C07259=1059.763,-17.708,-67.702,171.487,27.976,155.219
C07260=1059.770,-17.459,-67.715,171.489,27.977,155.219
C07261=1059.775,-17.210,-67.729,171.490,27.980,155.219
C07262=1059.782,-16.960,-67.743,171.492,27.982,155.219
C07263=1059.788,-16.710,-67.756,171.493,27.984,155.220
C07264=1059.794,-16.461,-67.771,171.495,27.986,155.220
C07265=1059.801,-16.211,-67.784,171.497,27.989,155.220
C07266=1059.806,-15.962,-67.798,171.498,27.991,155.220
C07267=1059.813,-15.712,-67.812,171.500,27.993,155.221
C07268=1059.818,-15.462,-67.825,171.502,27.995,155.221
C07269=1059.825,-15.214,-67.839,171.502,27.997,155.221
C07270=1059.831,-14.963,-67.854,171.504,27.999,155.221
C07271=1059.837,-14.714,-67.867,171.506,28.002,155.222
C07272=1059.843,-14.464,-67.881,171.507,28.004,155.222
C07273=1059.850,-14.215,-67.895,171.509,28.006,155.222
C07274=1059.855,-13.966,-67.909,171.510,28.009,155.223
C07275=1059.861,-13.715,-67.923,171.512,28.011,155.223
C07276=1059.868,-13.467,-67.937,171.514,28.013,155.223
C07277=1059.873,-13.217,-67.951,171.515,28.015,155.223
C07278=1059.880,-12.967,-67.965,171.517,28.018,155.224
C07279=1059.886,-12.718,-67.979,171.519,28.020,155.224
C07280=1059.892,-12.468,-67.994,171.520,28.022,155.224
C07281=1059.898,-12.219,-68.007,171.522,28.024,155.225
C07282=1059.904,-11.969,-68.021,171.523,28.026,155.225
C07283=1059.910,-11.719,-68.036,171.524,28.029,155.225
C07284=1059.916,-11.470,-68.049,171.526,28.031,155.225
C07285=1059.922,-11.220,-68.063,171.528,28.033,155.226
C07286=1059.928,-10.971,-68.078,171.529,28.035,155.226
C07287=1059.934,-10.722,-68.091,171.531,28.038,155.226
C07288=1059.941,-10.472,-68.106,171.532,28.040,155.226
C07289=1059.946,-10.222,-68.120,171.534,28.042,155.227
C07290=1059.953,-9.972,-68.133,171.536,28.045,155.227
C07291=1059.959,-9.723,-68.148,171.537,28.047,155.227
C07292=1059.965,-9.473,-68.162,171.539,28.049,155.228
C07293=1059.972,-9.225,-68.176,171.540,28.051,155.228
C07294=1059.977,-8.975,-68.190,171.541,28.054,155.228
C07295=1059.983,-8.725,-68.204,171.543,28.056,155.228
C07296=1059.990,-8.476,-68.218,171.545,28.058,155.229
C07297=1059.996,-8.226,-68.233,171.546,28.060,155.229
C07298=1060.001,-7.977,-68.247,171.548,28.063,155.229
C07299=1060.008,-7.727,-68.261,171.549,28.065,155.230
C07300=1060.014,-7.478,-68.275,171.551,28.067,155.230
C07301=1060.020,-7.228,-68.290,171.553,28.069,155.230
C07302=1060.027,-6.979,-68.304,171.554,28.072,155.230
C07303=1060.033,-6.729,-68.318,171.556,28.074,155.231
C07304=1060.039,-6.480,-68.332,171.557,28.076,155.231
C07305=1060.045,-6.229,-68.347,171.558,28.079,155.231
C07306=1060.051,-5.981,-68.361,171.560,28.081,155.232
C07307=1060.057,-5.731,-68.375,171.562,28.083,155.232
C07308=1060.063,-5.482,-68.389,171.563,28.085,155.232
C07309=1060.070,-5.232,-68.403,171.565,28.088,155.232
C07310=1060.076,-4.983,-68.418,171.566,28.090,155.233
C07311=1060.082,-4.732,-68.432,171.568,28.092,155.233
C07312=1060.088,-4.484,-68.446,171.570,28.094,155.233
C07313=1060.095,-4.234,-68.461,171.571,28.097,155.233
C07314=1060.101,-3.984,-68.475,171.573,28.099,155.234
C07315=1060.106,-3.735,-68.490,171.574,28.101,155.234
C07316=1060.113,-3.485,-68.503,171.575,28.104,155.234
C07317=1060.119,-3.236,-68.518,171.577,28.106,155.235
C07318=1060.125,-2.986,-68.533,171.579,28.108,155.235
C07319=1060.131,-2.737,-68.547,171.580,28.110,155.235
C07320=1060.137,-2.455,-68.563,171.582,28.113,155.236
C07321=1060.145,-2.174,-68.580,171.583,28.116,155.236
C07322=1060.151,-1.893,-68.596,171.585,28.118,155.236
C07323=1060.158,-1.612,-68.612,171.587,28.121,155.237
C07324=1060.164,-1.362,-68.627,171.588,28.123,155.237
C07325=1060.170,-1.113,-68.641,171.590,28.126,155.237
C07326=1060.176,-0.863,-68.656,171.591,28.128,155.238
C07327=1060.182,-0.614,-68.670,171.593,28.131,155.238
C07328=1060.188,-0.364,-68.685,171.595,28.134,155.238
C07329=1060.194,-0.114,-68.699,171.596,28.136,155.239
C07330=1060.200,0.135,-68.714,171.598,28.138,155.239
C07331=1060.207,0.385,-68.729,171.600,28.140,155.239
C07332=1060.212,0.634,-68.743,171.600,28.143,155.239
C07333=1060.218,0.884,-68.758,171.602,28.145,155.240
C07334=1060.224,1.133,-68.772,171.603,28.147,155.240
C07335=1060.231,1.383,-68.787,171.605,28.150,155.240
C07336=1060.236,1.632,-68.802,171.607,28.152,155.241
C07337=1060.243,1.882,-68.816,171.608,28.155,155.241
C07338=1060.248,2.131,-68.831,171.610,28.157,155.241
C07339=1060.254,2.381,-68.846,171.612,28.160,155.242
C07340=1060.260,2.630,-68.861,171.612,28.162,155.242
C07341=1060.266,2.879,-68.876,171.614,28.164,155.242
C07342=1060.272,3.130,-68.890,171.615,28.166,155.242
C07343=1060.278,3.379,-68.904,171.617,28.169,155.243
C07344=1060.284,3.628,-68.919,171.619,28.171,155.243
C07345=1060.291,3.878,-68.934,171.620,28.173,155.243
C07346=1060.297,4.127,-68.949,171.622,28.176,155.244
C07347=1060.303,4.377,-68.964,171.624,28.179,155.244
C07348=1060.309,4.626,-68.979,171.625,28.181,155.244
C07349=1060.315,4.876,-68.993,171.626,28.183,155.245
C07350=1060.321,5.125,-69.008,171.627,28.186,155.245
C07351=1060.327,5.374,-69.022,171.629,28.188,155.245
C07352=1060.333,5.624,-69.037,171.631,28.190,155.246
C07353=1060.340,5.874,-69.052,171.632,28.193,155.246
C07354=1060.345,6.123,-69.067,171.634,28.195,155.246
C07355=1060.352,6.372,-69.082,171.636,28.197,155.246
C07356=1060.358,6.622,-69.097,171.637,28.200,155.247
C07357=1060.364,6.871,-69.111,171.638,28.202,155.247
C07358=1060.370,7.121,-69.127,171.640,28.204,155.247
C07359=1060.376,7.371,-69.142,171.641,28.207,155.248
C07360=1060.382,7.620,-69.156,171.643,28.209,155.248
C07361=1060.388,7.870,-69.170,171.644,28.212,155.248
C07362=1060.394,8.119,-69.185,171.646,28.214,155.249
C07363=1060.400,8.368,-69.200,171.648,28.217,155.249
C07364=1060.406,8.618,-69.215,171.648,28.219,155.249
C07365=1060.413,8.868,-69.230,171.650,28.221,155.250
C07366=1060.419,9.117,-69.245,171.652,28.224,155.250
C07367=1060.425,9.366,-69.259,171.653,28.226,155.250
C07368=1060.431,9.616,-69.274,171.655,28.228,155.251
C07369=1060.438,9.866,-69.289,171.656,28.231,155.251
C07370=1060.444,10.115,-69.306,171.658,28.233,155.251
C07371=1060.450,10.364,-69.320,171.660,28.236,155.251
C07372=1060.456,10.614,-69.335,171.660,28.238,155.252
C07373=1060.462,10.863,-69.350,171.662,28.240,155.252
C07374=1060.468,11.112,-69.365,171.664,28.243,155.252
C07375=1060.474,11.362,-69.380,171.665,28.245,155.253
C07376=1060.481,11.612,-69.395,171.667,28.248,155.253
C07377=1060.487,11.861,-69.409,171.669,28.250,155.253
C07378=1060.493,12.111,-69.425,171.670,28.252,155.254
C07379=1060.499,12.360,-69.440,171.671,28.255,155.254
C07380=1060.505,12.610,-69.455,171.672,28.257,155.254
C07381=1060.511,12.859,-69.469,171.674,28.259,155.255
C07382=1060.518,13.109,-69.485,171.676,28.262,155.255
C07383=1060.524,13.357,-69.500,171.677,28.264,155.255
C07384=1060.531,13.642,-69.517,171.679,28.267,155.256
C07385=1060.538,13.925,-69.534,171.681,28.269,155.256
C07386=1060.546,14.208,-69.551,171.682,28.272,155.256
C07387=1060.552,14.491,-69.568,171.684,28.275,155.257
C07388=1060.559,14.740,-69.584,171.685,28.277,155.257
C07389=1060.564,14.990,-69.599,171.687,28.280,155.257
C07390=1060.570,15.239,-69.614,171.689,28.282,155.258
C07391=1060.576,15.489,-69.629,171.690,28.285,155.258
C07392=1060.582,15.739,-69.644,171.692,28.287,155.258
C07393=1060.588,15.987,-69.660,171.693,28.290,155.259
C07394=1060.595,16.237,-69.675,171.694,28.292,155.259
C07395=1060.600,16.487,-69.690,171.696,28.295,155.259
C07396=1060.607,16.737,-69.705,171.697,28.297,155.260
C07397=1060.613,16.986,-69.721,171.699,28.299,155.260
C07398=1060.618,17.235,-69.736,171.701,28.302,155.260
C07399=1060.625,17.485,-69.751,171.702,28.304,155.261
C07400=1060.631,17.734,-69.766,171.703,28.307,155.261
C07401=1060.637,17.984,-69.782,171.705,28.309,155.261
C07402=1060.643,18.233,-69.797,171.706,28.312,155.262
C07403=1060.648,18.483,-69.812,171.708,28.314,155.262
C07404=1060.655,18.732,-69.828,171.709,28.317,155.262
C07405=1060.662,18.981,-69.843,171.711,28.319,155.263
C07406=1060.667,19.231,-69.858,171.713,28.321,155.263
C07407=1060.674,19.480,-69.874,171.713,28.324,155.263
C07408=1060.680,19.730,-69.889,171.715,28.326,155.264
C07409=1060.685,19.979,-69.904,171.716,28.329,155.264
C07410=1060.692,20.228,-69.920,171.718,28.331,155.264
C07411=1060.698,20.478,-69.935,171.720,28.334,155.265
C07412=1060.704,20.728,-69.950,171.721,28.336,155.265
C07413=1060.710,20.977,-69.967,171.722,28.339,155.265
C07414=1060.716,21.227,-69.981,171.724,28.341,155.266
C07415=1060.722,21.476,-69.998,171.725,28.344,155.266
C07416=1060.728,21.725,-70.012,171.727,28.346,155.266
C07417=1060.734,21.974,-70.029,171.728,28.349,155.267
C07418=1060.740,22.224,-70.044,171.730,28.351,155.267
C07419=1060.746,22.474,-70.059,171.732,28.354,155.267
C07420=1060.753,22.723,-70.075,171.732,28.356,155.268
C07421=1060.758,22.973,-70.090,171.734,28.359,155.268
C07422=1060.765,23.222,-70.106,171.736,28.361,155.268
C07423=1060.770,23.471,-70.121,171.737,28.364,155.269
C07424=1060.777,23.720,-70.137,171.739,28.366,155.269
C07425=1060.782,23.970,-70.152,171.741,28.369,155.269
C07426=1060.789,24.219,-70.168,171.741,28.371,155.270
C07427=1060.795,24.469,-70.184,171.743,28.374,155.270
C07428=1060.801,24.718,-70.199,171.744,28.376,155.270
C07429=1060.807,24.968,-70.215,171.746,28.379,155.271
C07430=1060.814,25.217,-70.230,171.748,28.381,155.271
C07431=1060.819,25.467,-70.246,171.749,28.384,155.271
C07432=1060.825,25.717,-70.262,171.750,28.386,155.272
C07433=1060.831,25.966,-70.277,171.752,28.388,155.272
C07434=1060.837,26.215,-70.293,171.753,28.391,155.272
C07435=1060.844,26.465,-70.308,171.755,28.393,155.273
C07436=1060.849,26.714,-70.324,171.756,28.396,155.273
C07437=1060.856,26.963,-70.340,171.758,28.398,155.273
C07438=1060.862,27.213,-70.355,171.759,28.400,155.274
C07439=1060.868,27.462,-70.372,171.760,28.403,155.274
C07440=1060.874,27.712,-70.387,171.762,28.406,155.275
C07441=1060.880,27.961,-70.403,171.764,28.408,155.275
C07442=1060.887,28.210,-70.419,171.765,28.411,155.275
C07443=1060.892,28.460,-70.434,171.767,28.413,155.275
C07444=1060.898,28.710,-70.450,171.768,28.416,155.276
C07445=1060.905,28.959,-70.466,171.769,28.418,155.276
C07446=1060.911,29.209,-70.482,171.771,28.421,155.277
C07447=1060.917,29.458,-70.498,171.772,28.423,155.277
C07448=1060.924,29.743,-70.515,171.774,28.426,155.277
C07449=1060.930,30.027,-70.534,171.776,28.429,155.278
C07450=1060.938,30.312,-70.551,171.777,28.432,155.278
C07451=1060.944,30.596,-70.570,171.779,28.435,155.279
C07452=1060.950,30.846,-70.586,171.780,28.438,155.279
C07453=1060.956,31.096,-70.602,171.782,28.440,155.279
C07454=1060.962,31.345,-70.617,171.784,28.443,155.280
C07455=1060.968,31.594,-70.634,171.785,28.445,155.280
C07456=1060.974,31.844,-70.649,171.786,28.447,155.280
C07457=1060.980,32.093,-70.666,171.787,28.450,155.281
C07458=1060.987,32.342,-70.681,171.789,28.452,155.281
C07459=1060.993,32.592,-70.697,171.791,28.455,155.281
C07460=1060.998,32.842,-70.713,171.792,28.458,155.282
C07461=1061.004,33.091,-70.729,171.794,28.460,155.282
C07462=1061.011,33.340,-70.745,171.795,28.463,155.282
C07463=1061.017,33.589,-70.761,171.796,28.465,155.283
C07464=1061.023,33.839,-70.777,171.798,28.468,155.283
C07465=1061.028,34.089,-70.793,171.799,28.470,155.283
C07466=1061.035,34.338,-70.809,171.801,28.473,155.284
C07467=1061.041,34.587,-70.825,171.803,28.476,155.284
C07468=1061.047,34.836,-70.841,171.803,28.478,155.284
C07469=1061.053,35.086,-70.857,171.805,28.480,155.285
C07470=1061.059,35.335,-70.874,171.807,28.483,155.285
C07471=1061.065,35.585,-70.889,171.808,28.485,155.286
C07472=1061.071,35.834,-70.905,171.810,28.488,155.286
C07473=1061.077,36.083,-70.921,171.812,28.490,155.286
C07474=1061.083,36.333,-70.937,171.812,28.493,155.287
C07475=1061.089,36.582,-70.954,171.814,28.495,155.287
C07476=1061.096,36.831,-70.969,171.815,28.498,155.287
C07477=1061.102,37.081,-70.986,171.817,28.501,155.288
C07478=1061.108,37.331,-71.002,171.819,28.503,155.288
C07479=1061.114,37.580,-71.018,171.820,28.506,155.288
C07480=1061.120,37.829,-71.035,171.821,28.508,155.289
C07481=1061.126,38.079,-71.050,171.823,28.511,155.289
C07482=1061.132,38.329,-71.066,171.824,28.513,155.289
C07483=1061.138,38.578,-71.083,171.826,28.516,155.290
C07484=1061.144,38.827,-71.099,171.827,28.518,155.290
C07485=1061.150,39.077,-71.115,171.828,28.521,155.291
C07486=1061.156,39.326,-71.132,171.830,28.523,155.291
C07487=1061.162,39.575,-71.148,171.831,28.526,155.291
C07488=1061.168,39.825,-71.164,171.833,28.529,155.292
C07489=1061.173,40.074,-71.180,171.835,28.532,155.292
C07490=1061.179,40.323,-71.197,171.836,28.534,155.292
C07491=1061.185,40.573,-71.213,171.837,28.536,155.293
C07492=1061.192,40.823,-71.229,171.838,28.539,155.293
C07493=1061.198,41.072,-71.246,171.840,28.541,155.293
C07494=1061.204,41.321,-71.263,171.842,28.544,155.294
C07495=1061.210,41.570,-71.279,171.843,28.547,155.294
C07496=1061.216,41.820,-71.295,171.844,28.549,155.294
C07497=1061.222,42.069,-71.311,171.846,28.552,155.295
C07498=1061.228,42.318,-71.328,171.847,28.555,155.295
C07499=1061.234,42.568,-71.344,171.849,28.557,155.296
C07500=1061.240,42.817,-71.360,171.851,28.560,155.296
C07501=1061.246,43.067,-71.377,171.852,28.562,155.296
C07502=1061.252,43.316,-71.393,171.853,28.564,155.297
C07503=1061.258,43.566,-71.409,171.854,28.567,155.297
C07504=1061.264,43.815,-71.426,171.856,28.570,155.297
C07505=1061.270,44.064,-71.443,171.858,28.573,155.298
C07506=1061.276,44.313,-71.459,171.859,28.575,155.298
C07507=1061.282,44.563,-71.476,171.860,28.577,155.299
C07508=1061.288,44.812,-71.492,171.862,28.580,155.299
C07509=1061.294,45.062,-71.509,171.863,28.583,155.299
C07510=1061.300,45.312,-71.525,171.865,28.586,155.300
C07511=1061.306,45.561,-71.542,171.866,28.588,155.300
C07512=1061.312,45.845,-71.561,171.868,28.591,155.300
C07513=1061.319,46.130,-71.580,171.870,28.594,155.301
C07514=1061.326,46.414,-71.599,171.871,28.597,155.301
C07515=1061.333,46.699,-71.618,171.873,28.600,155.302
C07516=1061.339,46.948,-71.634,171.874,28.603,155.302
C07517=1061.344,47.198,-71.651,171.876,28.605,155.302
C07518=1061.350,47.447,-71.668,171.877,28.608,155.303
C07519=1061.356,47.696,-71.684,171.878,28.611,155.303
C07520=1061.362,47.946,-71.701,171.880,28.613,155.304
C07521=1061.368,48.196,-71.717,171.881,28.616,155.304
C07522=1061.374,48.444,-71.734,171.883,28.618,155.304
C07523=1061.380,48.694,-71.751,171.885,28.621,155.305
C07524=1061.385,48.943,-71.767,171.885,28.624,155.305
C07525=1061.392,49.192,-71.784,171.887,28.627,155.306
C07526=1061.398,49.442,-71.801,171.889,28.629,155.306
C07527=1061.404,49.691,-71.817,171.890,28.632,155.306
C07528=1061.410,49.940,-71.835,171.892,28.634,155.307
C07529=1061.416,50.190,-71.851,171.892,28.637,155.307
C07530=1061.422,50.439,-71.867,171.894,28.639,155.307
C07531=1061.428,50.689,-71.885,171.896,28.642,155.308
C07532=1061.434,50.938,-71.902,171.897,28.645,155.308
C07533=1061.440,51.188,-71.918,171.899,28.647,155.309
C07534=1061.445,51.437,-71.935,171.900,28.650,155.309
C07535=1061.452,51.687,-71.952,171.901,28.652,155.309
C07536=1061.458,51.935,-71.969,171.903,28.655,155.310
C07537=1061.464,52.185,-71.985,171.905,28.658,155.310
C07538=1061.469,52.434,-72.002,171.906,28.661,155.310
C07539=1061.475,52.683,-72.019,171.908,28.663,155.311
C07540=1061.482,52.933,-72.036,171.908,28.665,155.311
C07541=1061.487,53.182,-72.053,171.910,28.668,155.311
C07542=1061.493,53.432,-72.070,171.912,28.671,155.312
C07543=1061.500,53.681,-72.087,171.913,28.673,155.312
C07544=1061.505,53.931,-72.104,171.915,28.676,155.313
C07545=1061.512,54.179,-72.121,171.916,28.678,155.313
C07546=1061.518,54.429,-72.137,171.917,28.681,155.313
C07547=1061.523,54.679,-72.154,171.919,28.683,155.314
C07548=1061.530,54.928,-72.171,171.921,28.686,155.314
C07549=1061.536,55.177,-72.187,171.922,28.689,155.314
C07550=1061.542,55.427,-72.205,171.924,28.692,155.315
C07551=1061.548,55.676,-72.222,171.924,28.694,155.315
C07552=1061.554,55.925,-72.239,171.926,28.697,155.316
C07553=1061.560,56.174,-72.256,171.928,28.699,155.316
C07554=1061.566,56.424,-72.273,171.929,28.702,155.316
C07555=1061.572,56.673,-72.290,171.931,28.704,155.317
C07556=1061.578,56.923,-72.307,171.932,28.707,155.317
C07557=1061.584,57.172,-72.324,171.933,28.710,155.317
C07558=1061.590,57.421,-72.340,171.935,28.712,155.318
C07559=1061.596,57.670,-72.358,171.937,28.715,155.318
C07560=1061.602,57.920,-72.374,171.938,28.717,155.319
C07561=1061.608,58.169,-72.392,171.940,28.720,155.319
C07562=1061.614,58.418,-72.409,171.940,28.723,155.319
C07563=1061.621,58.668,-72.426,171.942,28.725,155.320
C07564=1061.626,58.917,-72.443,171.944,28.728,155.320
C07565=1061.633,59.167,-72.460,171.945,28.730,155.320
C07566=1061.639,59.416,-72.477,171.947,28.733,155.321
C07567=1061.645,59.665,-72.494,171.948,28.735,155.321
C07568=1061.651,59.915,-72.511,171.949,28.738,155.322
C07569=1061.657,60.164,-72.528,171.951,28.741,155.322
C07570=1061.664,60.414,-72.546,171.953,28.743,155.322
C07571=1061.669,60.663,-72.562,171.954,28.746,155.323
C07572=1061.675,60.912,-72.580,171.956,28.748,155.323
C07573=1061.682,61.161,-72.597,171.957,28.750,155.323
C07574=1061.688,61.411,-72.613,171.958,28.753,155.324
C07575=1061.694,61.660,-72.631,171.960,28.756,155.324
C07576=1061.701,61.944,-72.650,171.961,28.759,155.324
C07577=1061.708,62.228,-72.670,171.963,28.762,155.325
C07578=1061.715,62.514,-72.690,171.965,28.765,155.325
C07579=1061.721,62.797,-72.709,171.966,28.768,155.326
C07580=1061.728,63.047,-72.726,171.968,28.770,155.326
C07581=1061.734,63.296,-72.744,171.970,28.773,155.326
C07582=1061.740,63.546,-72.761,171.971,28.775,155.327
C07583=1061.747,63.794,-72.778,171.973,28.778,155.327
C07584=1061.753,64.044,-72.796,171.974,28.780,155.328
C07585=1061.759,64.293,-72.812,171.975,28.783,155.328
C07586=1061.765,64.543,-72.830,171.977,28.786,155.328
C07587=1061.770,64.792,-72.847,171.978,28.788,155.329
C07588=1061.776,65.041,-72.864,171.980,28.791,155.329
C07589=1061.783,65.291,-72.882,171.982,28.793,155.329
C07590=1061.789,65.539,-72.899,171.982,28.796,155.330
C07591=1061.795,65.789,-72.917,171.984,28.799,155.330
C07592=1061.800,66.039,-72.934,171.986,28.802,155.331
C07593=1061.807,66.288,-72.951,171.987,28.804,155.331
C07594=1061.813,66.537,-72.969,171.989,28.806,155.331
C07595=1061.818,66.786,-72.986,171.991,28.809,155.332
C07596=1061.825,67.036,-73.004,171.991,28.812,155.332
C07597=1061.830,67.285,-73.021,171.993,28.815,155.333
C07598=1061.837,67.535,-73.039,171.994,28.817,155.333
C07599=1061.843,67.783,-73.056,171.996,28.820,155.333
C07600=1061.849,68.033,-73.074,171.998,28.822,155.334
C07601=1061.854,68.283,-73.091,171.999,28.825,155.334
C07602=1061.860,68.532,-73.109,172.000,28.828,155.334
C07603=1061.867,68.781,-73.126,172.002,28.830,155.335
C07604=1061.873,69.031,-73.144,172.003,28.833,155.335
C07605=1061.878,69.280,-73.161,172.005,28.835,155.336
C07606=1061.885,69.529,-73.179,172.007,28.838,155.336
C07607=1061.891,69.778,-73.196,172.007,28.841,155.336
C07608=1061.897,70.028,-73.214,172.009,28.843,155.337
C07609=1061.902,70.277,-73.232,172.010,28.846,155.337
C07610=1061.908,70.526,-73.249,172.012,28.848,155.337
C07611=1061.915,70.776,-73.267,172.014,28.851,155.338
C07612=1061.920,71.025,-73.284,172.015,28.854,155.338
C07613=1061.926,71.274,-73.302,172.016,28.856,155.339
C07614=1061.932,71.523,-73.320,172.018,28.859,155.339
C07615=1061.938,71.773,-73.338,172.019,28.862,155.339
C07616=1061.944,72.022,-73.355,172.021,28.865,155.340
C07617=1061.950,72.272,-73.373,172.023,28.867,155.340
C07618=1061.956,72.520,-73.391,172.024,28.870,155.341
C07619=1061.962,72.770,-73.409,172.025,28.872,155.341
C07620=1061.968,73.019,-73.426,172.027,28.875,155.341
C07621=1061.974,73.269,-73.444,172.028,28.878,155.342
C07622=1061.979,73.518,-73.462,172.030,28.881,155.342
C07623=1061.986,73.767,-73.479,172.031,28.883,155.343
C07624=1061.992,74.016,-73.497,172.032,28.886,155.343
C07625=1061.998,74.266,-73.515,172.034,28.888,155.343
C07626=1062.004,74.516,-73.533,172.035,28.891,155.344
C07627=1062.010,74.764,-73.551,172.037,28.894,155.344
C07628=1062.016,75.014,-73.569,172.039,28.896,155.344
C07629=1062.021,75.263,-73.586,172.040,28.899,155.345
C07630=1062.028,75.513,-73.604,172.041,28.902,155.345
C07631=1062.034,75.761,-73.621,172.043,28.904,155.346
C07632=1062.040,76.011,-73.639,172.044,28.907,155.346
C07633=1062.046,76.259,-73.658,172.046,28.909,155.346
C07634=1062.052,76.509,-73.676,172.048,28.912,155.347
C07635=1062.058,76.759,-73.693,172.049,28.915,155.347
C07636=1062.064,77.008,-73.711,172.050,28.917,155.348
C07637=1062.070,77.258,-73.729,172.052,28.920,155.348
C07638=1062.075,77.506,-73.747,172.053,28.922,155.348
C07639=1062.082,77.756,-73.765,172.055,28.925,155.349
C07640=1062.088,78.040,-73.785,172.056,28.928,155.349
C07641=1062.096,78.324,-73.806,172.058,28.931,155.350
C07642=1062.102,78.608,-73.826,172.060,28.934,155.350
C07643=1062.109,78.892,-73.847,172.061,28.937,155.351
C07644=1062.115,79.142,-73.865,172.063,28.940,155.351
C07645=1062.121,79.391,-73.882,172.065,28.943,155.351
C07646=1062.126,79.641,-73.901,172.066,28.946,155.352
C07647=1062.132,79.890,-73.920,172.068,28.948,155.352
C07648=1062.138,80.139,-73.937,172.068,28.951,155.353
C07649=1062.144,80.389,-73.955,172.070,28.953,155.353
C07650=1062.150,80.637,-73.973,172.072,28.956,155.353
C07651=1062.156,80.887,-73.991,172.073,28.959,155.354
C07652=1062.162,81.135,-74.010,172.075,28.961,155.354
C07653=1062.168,81.385,-74.027,172.077,28.964,155.354
C07654=1062.173,81.635,-74.046,172.077,28.967,155.355
C07655=1062.179,81.884,-74.064,172.079,28.969,155.355
C07656=1062.185,82.133,-74.082,172.081,28.972,155.356
C07657=1062.191,82.383,-74.100,172.082,28.975,155.356
C07658=1062.197,82.631,-74.118,172.084,28.978,155.356
C07659=1062.203,82.881,-74.136,172.086,28.980,155.357
C07660=1062.209,83.130,-74.155,172.086,28.983,155.357
C07661=1062.215,83.380,-74.173,172.088,28.985,155.358
C07662=1062.221,83.629,-74.192,172.090,28.988,155.358
C07663=1062.227,83.878,-74.209,172.091,28.991,155.358
C07664=1062.233,84.128,-74.227,172.093,28.993,155.359
C07665=1062.239,84.377,-74.246,172.095,28.996,155.359
C07666=1062.245,84.626,-74.264,172.095,28.999,155.360
C07667=1062.250,84.875,-74.283,172.097,29.001,155.360
C07668=1062.256,85.125,-74.301,172.098,29.004,155.360
C07669=1062.262,85.373,-74.319,172.100,29.007,155.361
C07670=1062.268,85.623,-74.337,172.102,29.009,155.361
C07671=1062.275,85.872,-74.356,172.103,29.012,155.361
C07672=1062.280,86.121,-74.373,172.105,29.015,155.362
C07673=1062.286,86.371,-74.392,172.106,29.017,155.362
C07674=1062.292,86.620,-74.410,172.107,29.020,155.363
C07675=1062.299,86.870,-74.429,172.109,29.023,155.363
C07676=1062.304,87.118,-74.447,172.111,29.025,155.364
C07677=1062.310,87.368,-74.465,172.112,29.028,155.364
C07678=1062.317,87.617,-74.484,172.114,29.030,155.364
C07679=1062.322,87.866,-74.502,172.116,29.033,155.365
C07680=1062.328,88.115,-74.521,172.116,29.036,155.365
C07681=1062.334,88.365,-74.539,172.118,29.038,155.365
C07682=1062.341,88.614,-74.557,172.120,29.041,155.366
C07683=1062.346,88.863,-74.575,172.121,29.044,155.366
C07684=1062.352,89.113,-74.594,172.123,29.047,155.367
C07685=1062.358,89.362,-74.613,172.125,29.049,155.367
C07686=1062.365,89.611,-74.631,172.125,29.051,155.367
C07687=1062.370,89.860,-74.649,172.127,29.054,155.368
C07688=1062.376,90.109,-74.668,172.129,29.057,155.368
C07689=1062.382,90.358,-74.687,172.130,29.060,155.369
C07690=1062.388,90.608,-74.705,172.132,29.062,155.369
C07691=1062.394,90.857,-74.723,172.134,29.065,155.369
C07692=1062.400,91.106,-74.742,172.135,29.068,155.370
C07693=1062.406,91.356,-74.760,172.136,29.070,155.370
C07694=1062.412,91.605,-74.779,172.138,29.073,155.371
C07695=1062.418,91.854,-74.798,172.139,29.076,155.371
C07696=1062.424,92.103,-74.816,172.141,29.078,155.371
C07697=1062.429,92.353,-74.835,172.143,29.081,155.372
C07698=1062.436,92.602,-74.854,172.144,29.084,155.372
C07699=1062.441,92.851,-74.872,172.146,29.086,155.372
C07700=1062.447,93.100,-74.890,172.147,29.089,155.373
C07701=1062.453,93.350,-74.910,172.148,29.092,155.373
C07702=1062.459,93.599,-74.928,172.150,29.094,155.374
C07703=1062.464,93.848,-74.947,172.151,29.097,155.374
C07704=1062.471,94.132,-74.968,172.153,29.100,155.375
C07705=1062.479,94.416,-74.989,172.155,29.103,155.375
C07706=1062.485,94.701,-75.011,172.156,29.107,155.376
C07707=1062.492,94.985,-75.032,172.158,29.109,155.376
C07708=1062.498,95.234,-75.051,172.160,29.112,155.376
C07709=1062.504,95.482,-75.070,172.161,29.115,155.377
C07710=1062.509,95.732,-75.088,172.163,29.117,155.377
C07711=1062.515,95.982,-75.107,172.164,29.120,155.378
C07712=1062.521,96.231,-75.126,172.166,29.123,155.378
C07713=1062.527,96.480,-75.145,172.168,29.126,155.378
C07714=1062.533,96.729,-75.164,172.169,29.128,155.379
C07715=1062.539,96.978,-75.182,172.170,29.131,155.379
C07716=1062.545,97.227,-75.201,172.172,29.133,155.379
C07717=1062.551,97.477,-75.220,172.174,29.136,155.380
C07718=1062.557,97.726,-75.239,172.175,29.139,155.380
C07719=1062.563,97.976,-75.257,172.177,29.141,155.381
C07720=1062.569,98.225,-75.277,172.178,29.144,155.381
C07721=1062.574,98.474,-75.295,172.180,29.147,155.381
C07722=1062.580,98.723,-75.314,172.182,29.150,155.382
C07723=1062.587,98.972,-75.333,172.182,29.152,155.382
C07724=1062.592,99.222,-75.352,172.184,29.155,155.383
C07725=1062.599,99.471,-75.371,172.186,29.158,155.383
C07726=1062.604,99.720,-75.390,172.187,29.160,155.384
C07727=1062.611,99.969,-75.408,172.189,29.163,155.384
C07728=1062.616,100.219,-75.428,172.191,29.165,155.384
C07729=1062.622,100.467,-75.446,172.192,29.168,155.385
C07730=1062.628,100.717,-75.465,172.194,29.171,155.385
C07731=1062.634,100.966,-75.484,172.195,29.173,155.385
C07732=1062.640,101.215,-75.503,172.196,29.176,155.386
C07733=1062.646,101.465,-75.522,172.198,29.179,155.386
C07734=1062.652,101.714,-75.541,172.200,29.182,155.387
C07735=1062.658,101.963,-75.560,172.201,29.184,155.387
C07736=1062.664,102.213,-75.580,172.203,29.187,155.387
C07737=1062.669,102.461,-75.599,172.205,29.190,155.388
C07738=1062.675,102.710,-75.618,172.206,29.192,155.388
C07739=1062.681,102.959,-75.637,172.207,29.195,155.389
C07740=1062.687,103.209,-75.656,172.209,29.198,155.389
C07741=1062.692,103.458,-75.676,172.210,29.200,155.390
C07742=1062.699,103.707,-75.694,172.212,29.203,155.390
C07743=1062.705,103.957,-75.713,172.214,29.206,155.390
C07744=1062.710,104.206,-75.733,172.215,29.209,155.391
C07745=1062.716,104.455,-75.753,172.217,29.211,155.391
C07746=1062.723,104.704,-75.771,172.219,29.214,155.392
C07747=1062.728,104.953,-75.790,172.220,29.217,155.392
C07748=1062.733,105.202,-75.809,172.221,29.219,155.392
C07749=1062.739,105.452,-75.829,172.223,29.222,155.393
C07750=1062.746,105.701,-75.847,172.224,29.225,155.393
C07751=1062.752,105.949,-75.867,172.226,29.228,155.394
C07752=1062.757,106.199,-75.886,172.228,29.230,155.394
C07753=1062.763,106.448,-75.906,172.229,29.233,155.394
C07754=1062.769,106.697,-75.924,172.231,29.235,155.395
C07755=1062.775,106.946,-75.944,172.233,29.238,155.395
C07756=1062.781,107.196,-75.964,172.234,29.241,155.395
C07757=1062.787,107.445,-75.983,172.235,29.243,155.396
C07758=1062.792,107.695,-76.002,172.237,29.246,155.396
C07759=1062.799,107.943,-76.021,172.238,29.249,155.397
C07760=1062.805,108.193,-76.041,172.240,29.251,155.397
C07761=1062.811,108.442,-76.060,172.242,29.254,155.398
C07762=1062.816,108.691,-76.079,172.243,29.257,155.398
C07763=1062.823,108.940,-76.099,172.245,29.260,155.398
C07764=1062.829,109.189,-76.118,172.247,29.262,155.399
C07765=1062.834,109.439,-76.137,172.248,29.265,155.399
C07766=1062.840,109.688,-76.157,172.250,29.268,155.400
C07767=1062.846,109.937,-76.176,172.251,29.270,155.400
C07768=1062.853,110.221,-76.199,172.253,29.273,155.400
C07769=1062.860,110.505,-76.220,172.255,29.277,155.401
C07770=1062.867,110.789,-76.242,172.257,29.279,155.401
C07771=1062.874,111.074,-76.264,172.258,29.283,155.402
C07772=1062.879,111.323,-76.284,172.260,29.285,155.402
C07773=1062.885,111.572,-76.303,172.262,29.288,155.402
C07774=1062.891,111.821,-76.323,172.263,29.290,155.403
C07775=1062.897,112.070,-76.343,172.265,29.293,155.403
C07776=1062.903,112.319,-76.363,172.267,29.296,155.404
C07777=1062.909,112.569,-76.382,172.268,29.298,155.404
C07778=1062.914,112.818,-76.401,172.270,29.301,155.405
C07779=1062.920,113.067,-76.421,172.272,29.304,155.405
C07780=1062.926,113.316,-76.440,172.272,29.306,155.405
C07781=1062.932,113.565,-76.460,172.274,29.309,155.406
C07782=1062.938,113.814,-76.479,172.276,29.312,155.406
C07783=1062.944,114.063,-76.499,172.277,29.315,155.407
C07784=1062.949,114.313,-76.519,172.279,29.317,155.407
C07785=1062.955,114.562,-76.539,172.281,29.320,155.407
C07786=1062.961,114.811,-76.558,172.282,29.323,155.408
C07787=1062.967,115.060,-76.578,172.284,29.326,155.408
C07788=1062.973,115.309,-76.597,172.286,29.329,155.409
C07789=1062.979,115.558,-76.617,172.287,29.332,155.409
C07790=1062.984,115.808,-76.637,172.289,29.334,155.410
C07791=1062.990,116.057,-76.657,172.291,29.337,155.410
C07792=1062.996,116.306,-76.677,172.291,29.340,155.410
C07793=1063.001,116.555,-76.696,172.293,29.342,155.411
C07794=1063.007,116.804,-76.716,172.295,29.345,155.411
C07795=1063.013,117.053,-76.735,172.296,29.348,155.412
C07796=1063.018,117.302,-76.756,172.298,29.350,155.412
C07797=1063.024,117.551,-76.776,172.300,29.353,155.412
C07798=1063.030,117.801,-76.795,172.301,29.356,155.413
C07799=1063.036,118.050,-76.815,172.303,29.359,155.413
C07800=1063.042,118.299,-76.835,172.305,29.361,155.414
C07801=1063.047,118.549,-76.855,172.306,29.364,155.414
C07802=1063.053,118.797,-76.875,172.308,29.367,155.414
C07803=1063.059,119.046,-76.895,172.310,29.370,155.415
C07804=1063.065,119.296,-76.914,172.311,29.373,155.415
C07805=1063.071,119.545,-76.934,172.312,29.375,155.416
C07806=1063.076,119.794,-76.955,172.314,29.378,155.416
C07807=1063.082,120.043,-76.974,172.315,29.381,155.417
C07808=1063.088,120.292,-76.994,172.317,29.384,155.417
C07809=1063.095,120.541,-77.014,172.319,29.386,155.417
C07810=1063.100,120.791,-77.035,172.320,29.389,155.418
C07811=1063.106,121.040,-77.054,172.322,29.392,155.418
C07812=1063.112,121.289,-77.074,172.324,29.394,155.419
C07813=1063.118,121.538,-77.094,172.325,29.397,155.419
C07814=1063.123,121.787,-77.115,172.327,29.400,155.419
C07815=1063.128,122.036,-77.134,172.329,29.403,155.420
C07816=1063.135,122.286,-77.154,172.330,29.405,155.420
C07817=1063.141,122.534,-77.174,172.332,29.408,155.421
C07818=1063.147,122.783,-77.194,172.334,29.411,155.421
C07819=1063.152,123.032,-77.215,172.335,29.413,155.421
C07820=1063.158,123.282,-77.234,172.337,29.416,155.422
C07821=1063.164,123.531,-77.254,172.339,29.419,155.422
C07822=1063.171,123.780,-77.274,172.340,29.422,155.423
C07823=1063.176,124.029,-77.295,172.342,29.424,155.423
C07824=1063.182,124.278,-77.315,172.344,29.427,155.423
C07825=1063.188,124.527,-77.335,172.344,29.430,155.424
C07826=1063.193,124.777,-77.354,172.346,29.432,155.424
C07827=1063.199,125.026,-77.375,172.348,29.435,155.425
C07828=1063.205,125.275,-77.395,172.350,29.438,155.425
C07829=1063.211,125.524,-77.415,172.351,29.440,155.426
C07830=1063.217,125.773,-77.435,172.353,29.443,155.426
C07831=1063.223,126.022,-77.455,172.355,29.446,155.426
C07832=1063.230,126.306,-77.478,172.357,29.449,155.427
C07833=1063.237,126.590,-77.502,172.359,29.452,155.427
C07834=1063.244,126.875,-77.525,172.360,29.455,155.428
C07835=1063.249,127.158,-77.548,172.362,29.458,155.428
C07836=1063.255,127.407,-77.567,172.364,29.461,155.429
C07837=1063.262,127.657,-77.588,172.365,29.464,155.429
C07838=1063.268,127.906,-77.608,172.367,29.466,155.429
C07839=1063.273,128.155,-77.628,172.369,29.469,155.430
C07840=1063.280,128.404,-77.649,172.371,29.472,155.430
C07841=1063.286,128.653,-77.669,172.372,29.474,155.431
C07842=1063.291,128.902,-77.689,172.374,29.477,155.431
C07843=1063.297,129.151,-77.709,172.376,29.480,155.431
C07844=1063.304,129.401,-77.729,172.377,29.483,155.432
C07845=1063.309,129.650,-77.750,172.379,29.485,155.432
C07846=1063.315,129.898,-77.770,172.381,29.487,155.433
C07847=1063.322,130.148,-77.790,172.382,29.490,155.433
C07848=1063.327,130.397,-77.811,172.384,29.493,155.433
C07849=1063.333,130.646,-77.831,172.386,29.496,155.434
C07850=1063.339,130.895,-77.851,172.387,29.498,155.434
C07851=1063.345,131.144,-77.872,172.389,29.501,155.435
C07852=1063.351,131.393,-77.892,172.391,29.504,155.435
C07853=1063.358,131.642,-77.913,172.392,29.506,155.435
C07854=1063.363,131.891,-77.933,172.394,29.509,155.436
C07855=1063.369,132.140,-77.953,172.396,29.512,155.436
C07856=1063.375,132.390,-77.974,172.397,29.515,155.437
C07857=1063.381,132.639,-77.994,172.399,29.517,155.437
C07858=1063.386,132.888,-78.015,172.401,29.520,155.437
C07859=1063.392,133.136,-78.035,172.403,29.523,155.438
C07860=1063.398,133.386,-78.056,172.404,29.525,155.438
C07861=1063.403,133.635,-78.077,172.406,29.528,155.439
C07862=1063.409,133.884,-78.097,172.408,29.531,155.439
C07863=1063.415,134.134,-78.118,172.409,29.534,155.440
C07864=1063.421,134.382,-78.138,172.411,29.537,155.440
C07865=1063.427,134.631,-78.159,172.413,29.540,155.440
C07866=1063.433,134.881,-78.180,172.414,29.542,155.441
C07867=1063.439,135.130,-78.200,172.416,29.545,155.441
C07868=1063.444,135.378,-78.221,172.418,29.548,155.442
C07869=1063.451,135.628,-78.241,172.419,29.550,155.442
C07870=1063.456,135.877,-78.262,172.421,29.553,155.442
C07871=1063.462,136.125,-78.283,172.423,29.556,155.443
C07872=1063.468,136.375,-78.303,172.424,29.559,155.443
C07873=1063.473,136.624,-78.324,172.426,29.561,155.444
C07874=1063.480,136.874,-78.344,172.428,29.564,155.444
C07875=1063.486,137.122,-78.366,172.429,29.567,155.444
C07876=1063.491,137.371,-78.386,172.431,29.569,155.445
C07877=1063.498,137.620,-78.407,172.433,29.572,155.445
C07878=1063.503,137.869,-78.428,172.435,29.575,155.446
C07879=1063.508,138.118,-78.448,172.436,29.577,155.446
C07880=1063.515,138.367,-78.469,172.438,29.580,155.447
C07881=1063.520,138.616,-78.490,172.440,29.583,155.447
C07882=1063.526,138.866,-78.511,172.441,29.586,155.447
C07883=1063.532,139.115,-78.532,172.443,29.589,155.448
C07884=1063.538,139.363,-78.552,172.446,29.592,155.448
C07885=1063.544,139.613,-78.574,172.447,29.594,155.449
C07886=1063.549,139.862,-78.594,172.449,29.597,155.449
C07887=1063.556,140.111,-78.615,172.451,29.600,155.449
C07888=1063.561,140.360,-78.636,172.452,29.603,155.450
C07889=1063.567,140.610,-78.657,172.454,29.605,155.450
C07890=1063.573,140.858,-78.678,172.456,29.608,155.451
C07891=1063.578,141.107,-78.699,172.457,29.611,155.451
C07892=1063.585,141.356,-78.720,172.459,29.613,155.452
C07893=1063.590,141.605,-78.740,172.461,29.616,155.452
C07894=1063.596,141.854,-78.762,172.462,29.619,155.452
C07895=1063.602,142.104,-78.782,172.464,29.622,155.453
C07896=1063.608,142.388,-78.806,172.466,29.625,155.453
C07897=1063.615,142.672,-78.830,172.468,29.628,155.454
C07898=1063.622,142.956,-78.854,172.470,29.632,155.454
C07899=1063.628,143.239,-78.878,172.472,29.634,155.455
C07900=1063.634,143.488,-78.900,172.473,29.637,155.455
C07901=1063.640,143.737,-78.921,172.475,29.640,155.456
C07902=1063.645,143.987,-78.942,172.477,29.643,155.456
C07903=1063.651,144.235,-78.963,172.479,29.646,155.456
C07904=1063.658,144.485,-78.983,172.481,29.649,155.457
C07905=1063.663,144.733,-79.005,172.483,29.651,155.457
C07906=1063.669,144.982,-79.026,172.485,29.654,155.458
C07907=1063.675,145.231,-79.047,172.486,29.657,155.458
C07908=1063.681,145.481,-79.069,172.488,29.659,155.458
C07909=1063.686,145.730,-79.089,172.490,29.662,155.459
C07910=1063.692,145.979,-79.111,172.491,29.665,155.459
C07911=1063.698,146.228,-79.132,172.493,29.667,155.460
C07912=1063.705,146.476,-79.153,172.495,29.671,155.460
C07913=1063.710,146.726,-79.174,172.496,29.673,155.461
C07914=1063.716,146.975,-79.195,172.498,29.676,155.461
C07915=1063.722,147.223,-79.217,172.500,29.679,155.461
C07916=1063.728,147.473,-79.237,172.502,29.681,155.462
C07917=1063.733,147.722,-79.259,172.504,29.684,155.462
C07918=1063.739,147.971,-79.280,172.506,29.687,155.463
C07919=1063.745,148.220,-79.302,172.508,29.690,155.463
C07920=1063.751,148.469,-79.323,172.509,29.692,155.463
C07921=1063.757,148.718,-79.344,172.511,29.695,155.464
C07922=1063.762,148.967,-79.365,172.513,29.698,155.464
C07923=1063.769,149.216,-79.387,172.514,29.701,155.465
C07924=1063.774,149.465,-79.408,172.516,29.704,155.465
C07925=1063.780,149.714,-79.429,172.518,29.707,155.466
C07926=1063.786,149.963,-79.451,172.519,29.709,155.466
C07927=1063.792,150.212,-79.472,172.521,29.712,155.466
C07928=1063.797,150.461,-79.493,172.523,29.715,155.467
C07929=1063.803,150.710,-79.515,172.526,29.718,155.467
C07930=1063.808,150.959,-79.536,172.527,29.721,155.468
C07931=1063.814,151.208,-79.558,172.529,29.723,155.468
C07932=1063.820,151.458,-79.579,172.531,29.726,155.469
C07933=1063.826,151.706,-79.601,172.532,29.729,155.469
C07934=1063.832,151.955,-79.622,172.534,29.732,155.469
C07935=1063.838,152.204,-79.644,172.536,29.734,155.470
C07936=1063.844,152.453,-79.665,172.537,29.738,155.470
C07937=1063.849,152.702,-79.687,172.539,29.740,155.471
C07938=1063.855,152.951,-79.709,172.541,29.743,155.471
C07939=1063.861,153.200,-79.730,172.543,29.746,155.472
C07940=1063.866,153.449,-79.752,172.545,29.748,155.472
C07941=1063.873,153.698,-79.773,172.547,29.751,155.472
C07942=1063.879,153.947,-79.795,172.549,29.754,155.473
C07943=1063.884,154.196,-79.816,172.550,29.757,155.473
C07944=1063.890,154.445,-79.838,172.552,29.760,155.474
C07945=1063.895,154.694,-79.860,172.554,29.762,155.474
C07946=1063.901,154.943,-79.881,172.555,29.765,155.475
C07947=1063.908,155.192,-79.903,172.558,29.768,155.475
C07948=1063.913,155.441,-79.924,172.560,29.771,155.475
C07949=1063.919,155.690,-79.946,172.561,29.774,155.476
C07950=1063.925,155.939,-79.968,172.563,29.777,155.476
C07951=1063.930,156.188,-79.989,172.565,29.779,155.477
C07952=1063.936,156.437,-80.011,172.566,29.782,155.477
C07953=1063.943,156.686,-80.033,172.568,29.785,155.478
C07954=1063.947,156.935,-80.055,172.570,29.787,155.478
C07955=1063.954,157.184,-80.076,172.572,29.791,155.478
C07956=1063.959,157.433,-80.097,172.574,29.794,155.479
C07957=1063.965,157.682,-80.120,172.576,29.796,155.479
C07958=1063.971,157.931,-80.142,172.578,29.799,155.480
C07959=1063.977,158.179,-80.163,172.579,29.802,155.480
C07960=1063.983,158.464,-80.188,172.582,29.805,155.481
C07961=1063.990,158.747,-80.213,172.584,29.808,155.481
C07962=1063.996,159.031,-80.238,172.586,29.812,155.482
C07963=1064.003,159.314,-80.263,172.588,29.815,155.482
C07964=1064.009,159.564,-80.284,172.590,29.818,155.483
C07965=1064.015,159.813,-80.307,172.591,29.820,155.483
C07966=1064.021,160.062,-80.329,172.593,29.823,155.483
C07967=1064.027,160.310,-80.350,172.596,29.826,155.484
C07968=1064.032,160.560,-80.372,172.597,29.829,155.484
C07969=1064.038,160.809,-80.394,172.599,29.831,155.485
C07970=1064.045,161.057,-80.416,172.601,29.835,155.485
C07971=1064.049,161.306,-80.438,172.603,29.837,155.486
C07972=1064.056,161.555,-80.460,172.604,29.840,155.486
C07973=1064.060,161.804,-80.482,172.607,29.843,155.486
C07974=1064.066,162.053,-80.505,172.609,29.846,155.487
C07975=1064.072,162.302,-80.526,172.610,29.849,155.487
C07976=1064.077,162.551,-80.548,172.612,29.852,155.488
C07977=1064.083,162.800,-80.571,172.614,29.855,155.488
C07978=1064.089,163.049,-80.593,172.615,29.857,155.489
C07979=1064.094,163.298,-80.615,172.618,29.861,155.489
C07980=1064.100,163.547,-80.638,172.620,29.864,155.490
C07981=1064.106,163.796,-80.659,172.621,29.867,155.490
C07982=1064.112,164.045,-80.682,172.623,29.870,155.491
C07983=1064.116,164.294,-80.704,172.625,29.872,155.491
C07984=1064.123,164.543,-80.726,172.626,29.875,155.491
C07985=1064.128,164.792,-80.749,172.629,29.878,155.492
C07986=1064.133,165.041,-80.770,172.631,29.881,155.492
C07987=1064.140,165.289,-80.793,172.633,29.884,155.493
C07988=1064.145,165.539,-80.815,172.634,29.887,155.493
C07989=1064.151,165.788,-80.838,172.636,29.890,155.494
C07990=1064.156,166.036,-80.859,172.638,29.893,155.494
C07991=1064.162,166.285,-80.882,172.640,29.896,155.495
C07992=1064.167,166.535,-80.904,172.642,29.898,155.495
C07993=1064.174,166.783,-80.927,172.644,29.902,155.496
C07994=1064.179,167.032,-80.949,172.645,29.904,155.496
C07995=1064.184,167.281,-80.972,172.647,29.907,155.496
C07996=1064.191,167.530,-80.993,172.650,29.910,155.497
C07997=1064.196,167.779,-81.016,172.652,29.913,155.497
C07998=1064.201,168.028,-81.038,172.653,29.916,155.498
C07999=1064.207,168.277,-81.061,172.655,29.919,155.498
C08000=1064.213,168.525,-81.083,172.657,29.922,155.499
C08001=1064.219,168.775,-81.106,172.659,29.925,155.499
C08002=1064.224,169.024,-81.128,172.661,29.928,155.500
C08003=1064.230,169.272,-81.150,172.663,29.931,155.500
C08004=1064.236,169.521,-81.173,172.664,29.934,155.500
C08005=1064.242,169.770,-81.196,172.667,29.937,155.501
C08006=1064.247,170.020,-81.218,172.669,29.939,155.501
C08007=1064.253,170.268,-81.240,172.670,29.943,155.502
C08008=1064.259,170.500,-81.261,172.672,29.945,155.502
C08009=1064.264,170.732,-81.282,172.674,29.948,155.503
C08010=1064.269,170.965,-81.303,172.676,29.951,155.503
C08011=1064.274,171.197,-81.324,172.677,29.953,155.503
C08012=1064.280,171.428,-81.345,172.679,29.956,155.504
C08013=1064.285,171.661,-81.366,172.681,29.959,155.504
C08014=1064.290,171.893,-81.387,172.684,29.962,155.505
C08015=1064.296,172.126,-81.408,172.685,29.964,155.505
C08016=1064.301,172.374,-81.431,172.687,29.967,155.506
C08017=1064.308,172.622,-81.453,172.689,29.970,155.506
C08018=1064.313,172.872,-81.476,172.690,29.973,155.506
C08019=1064.319,173.121,-81.498,172.693,29.976,155.507
C08020=1064.324,173.370,-81.521,172.695,29.978,155.507
C08021=1064.331,173.618,-81.544,172.696,29.982,155.508
C08022=1064.336,173.868,-81.566,172.698,29.984,155.508
C08023=1064.342,174.117,-81.589,172.701,29.987,155.509
C08024=1064.349,174.433,-81.618,172.703,29.991,155.509
C08025=1064.356,174.751,-81.647,172.705,29.994,155.510
C08026=1064.365,175.068,-81.675,172.708,29.998,155.510
C08027=1064.371,175.384,-81.704,172.710,30.002,155.511
C08028=1064.377,175.633,-81.727,172.712,30.005,155.511
C08029=1064.383,175.882,-81.750,172.715,30.008,155.512
C08030=1064.389,176.131,-81.772,172.716,30.011,155.512
C08031=1064.395,176.379,-81.795,172.718,30.014,155.513
C08032=1064.401,176.628,-81.818,172.721,30.017,155.513
C08033=1064.407,176.877,-81.841,172.723,30.019,155.514
C08034=1064.412,177.126,-81.864,172.724,30.023,155.514
C08035=1064.418,177.375,-81.887,172.726,30.025,155.515
C08036=1064.424,177.624,-81.909,172.729,30.028,155.515
C08037=1064.430,177.873,-81.932,172.730,30.031,155.515
C08038=1064.436,178.122,-81.955,172.732,30.034,155.516
C08039=1064.441,178.371,-81.978,172.735,30.037,155.516
C08040=1064.447,178.620,-82.000,172.737,30.040,155.517
C08041=1064.454,178.868,-82.023,172.738,30.043,155.517
C08042=1064.459,179.117,-82.046,172.740,30.045,155.518
C08043=1064.465,179.366,-82.069,172.743,30.048,155.518
C08044=1064.471,179.616,-82.092,172.744,30.051,155.519
C08045=1064.477,179.865,-82.115,172.746,30.054,155.519
C08046=1064.483,180.114,-82.138,172.749,30.057,155.519
C08047=1064.489,180.362,-82.160,172.750,30.060,155.520
C08048=1064.495,180.610,-82.184,172.752,30.063,155.520
C08049=1064.501,180.859,-82.207,172.755,30.066,155.521
C08050=1064.507,181.108,-82.230,172.757,30.069,155.521
C08051=1064.512,181.357,-82.253,172.758,30.072,155.522
C08052=1064.518,181.606,-82.276,172.761,30.075,155.522
C08053=1064.524,181.855,-82.299,172.763,30.078,155.523
C08054=1064.530,182.104,-82.322,172.764,30.080,155.523
C08055=1064.537,182.353,-82.344,172.767,30.083,155.523
C08056=1064.542,182.602,-82.367,172.769,30.086,155.524
C08057=1064.549,182.850,-82.391,172.771,30.089,155.524
C08058=1064.554,183.099,-82.414,172.773,30.092,155.525
C08059=1064.560,183.348,-82.437,172.775,30.095,155.525
C08060=1064.566,183.597,-82.460,172.777,30.098,155.526
C08061=1064.571,183.846,-82.483,172.779,30.101,155.526
C08062=1064.578,184.095,-82.506,172.781,30.103,155.526
C08063=1064.585,184.343,-82.529,172.783,30.107,155.527
C08064=1064.590,184.592,-82.552,172.786,30.109,155.527
C08065=1064.595,184.842,-82.576,172.787,30.113,155.528
C08066=1064.601,185.090,-82.599,172.789,30.115,155.528
C08067=1064.607,185.339,-82.622,172.792,30.119,155.529
C08068=1064.612,185.588,-82.646,172.793,30.121,155.529
C08069=1064.618,185.837,-82.669,172.795,30.125,155.530
C08070=1064.624,186.085,-82.692,172.798,30.128,155.530
C08071=1064.629,186.334,-82.716,172.799,30.131,155.531
C08072=1064.635,186.584,-82.739,172.801,30.134,155.531
C08073=1064.641,186.832,-82.763,172.804,30.137,155.532
C08074=1064.646,187.081,-82.786,172.806,30.140,155.532
C08075=1064.652,187.330,-82.809,172.807,30.143,155.533
C08076=1064.658,187.579,-82.833,172.810,30.146,155.533
C08077=1064.663,187.828,-82.857,172.812,30.149,155.534
C08078=1064.669,188.076,-82.880,172.813,30.152,155.534
C08079=1064.674,188.325,-82.904,172.816,30.155,155.535
C08080=1064.680,188.574,-82.927,172.818,30.158,155.535
C08081=1064.686,188.822,-82.950,172.820,30.161,155.536
C08082=1064.691,189.072,-82.974,172.822,30.165,155.536
C08083=1064.697,189.321,-82.998,172.824,30.167,155.536
C08084=1064.703,189.570,-83.021,172.827,30.171,155.537
C08085=1064.708,189.818,-83.045,172.828,30.173,155.537
C08086=1064.714,190.067,-83.068,172.830,30.177,155.538
C08087=1064.719,190.316,-83.092,172.833,30.180,155.538
C08088=1064.726,190.598,-83.119,172.835,30.183,155.539
C08089=1064.733,190.882,-83.146,172.837,30.187,155.540
C08090=1064.740,191.165,-83.173,172.840,30.190,155.540
C08091=1064.746,191.448,-83.200,172.842,30.194,155.541
C08092=1064.752,191.696,-83.223,172.844,30.197,155.541
C08093=1064.758,191.945,-83.247,172.846,30.200,155.542
C08094=1064.763,192.194,-83.270,172.849,30.203,155.542
C08095=1064.769,192.443,-83.294,172.850,30.206,155.543
C08096=1064.775,192.691,-83.319,172.853,30.209,155.543
C08097=1064.780,192.940,-83.341,172.855,30.212,155.543
C08098=1064.786,193.189,-83.366,172.856,30.215,155.544
C08099=1064.792,193.438,-83.390,172.859,30.218,155.544
C08100=1064.798,193.687,-83.413,172.861,30.221,155.545
C08101=1064.803,193.935,-83.437,172.863,30.225,155.545
C08102=1064.809,194.184,-83.461,172.865,30.227,155.546
C08103=1064.815,194.434,-83.485,172.868,30.231,155.546
C08104=1064.821,194.682,-83.508,172.870,30.234,155.547
C08105=1064.826,194.930,-83.532,172.871,30.237,155.547
C08106=1064.832,195.179,-83.555,172.874,30.240,155.548
C08107=1064.839,195.428,-83.579,172.876,30.243,155.548
C08108=1064.844,195.677,-83.604,172.878,30.246,155.549
C08109=1064.850,195.925,-83.627,172.880,30.249,155.549
C08110=1064.855,196.175,-83.651,172.883,30.252,155.550
C08111=1064.862,196.423,-83.675,172.885,30.255,155.550
C08112=1064.867,196.672,-83.699,172.886,30.258,155.551
C08113=1064.873,196.921,-83.723,172.889,30.261,155.551
C08114=1064.878,197.170,-83.747,172.891,30.265,155.552
C08115=1064.884,197.418,-83.770,172.893,30.267,155.552
C08116=1064.890,197.668,-83.795,172.895,30.271,155.553
C08117=1064.896,197.916,-83.819,172.898,30.274,155.553
C08118=1064.902,198.165,-83.843,172.900,30.277,155.554
C08119=1064.908,198.414,-83.867,172.902,30.280,155.554
C08120=1064.914,198.662,-83.891,172.904,30.283,155.555
C08121=1064.919,198.911,-83.914,172.907,30.286,155.555
C08122=1064.925,199.160,-83.939,172.908,30.289,155.556
C08123=1064.931,199.409,-83.962,172.910,30.292,155.556
C08124=1064.937,199.658,-83.987,172.913,30.295,155.557
C08125=1064.943,199.906,-84.011,172.915,30.299,155.557
C08126=1064.949,200.155,-84.035,172.917,30.301,155.557
C08127=1064.955,200.404,-84.059,172.919,30.305,155.558
C08128=1064.960,200.652,-84.083,172.922,30.308,155.558
C08129=1064.967,200.901,-84.107,172.923,30.311,155.559
C08130=1064.972,201.150,-84.132,172.926,30.314,155.559
C08131=1064.979,201.399,-84.156,172.928,30.317,155.560
C08132=1064.984,201.647,-84.180,172.931,30.320,155.560
C08133=1064.991,201.896,-84.204,172.932,30.323,155.561
C08134=1064.996,202.145,-84.228,172.935,30.326,155.561
C08135=1065.002,202.394,-84.252,172.937,30.329,155.562
C08136=1065.008,202.643,-84.276,172.939,30.333,155.562
C08137=1065.014,202.891,-84.301,172.941,30.336,155.563
C08138=1065.019,203.140,-84.325,172.944,30.339,155.563
C08139=1065.025,203.389,-84.350,172.946,30.342,155.564
C08140=1065.030,203.638,-84.374,172.948,30.345,155.564
C08141=1065.037,203.887,-84.398,172.950,30.349,155.565
C08142=1065.042,204.135,-84.423,172.953,30.352,155.565
C08143=1065.048,204.384,-84.447,172.954,30.355,155.566
C08144=1065.053,204.632,-84.472,172.957,30.359,155.566
C08145=1065.059,204.882,-84.496,172.959,30.361,155.567
C08146=1065.065,205.130,-84.520,172.961,30.365,155.567
C08147=1065.071,205.379,-84.545,172.963,30.368,155.568
C08148=1065.077,205.627,-84.570,172.966,30.371,155.568
C08149=1065.083,205.877,-84.594,172.968,30.374,155.569
C08150=1065.088,206.125,-84.618,172.970,30.378,155.570
C08151=1065.093,206.374,-84.643,172.972,30.380,155.570
C08152=1065.119,207.420,-84.746,173.131,30.459,155.576
C08153=1065.125,207.641,-84.768,173.133,30.463,155.576
C08154=1065.129,207.862,-84.791,173.135,30.467,155.577
C08155=1065.134,208.083,-84.813,173.137,30.470,155.578
C08156=1065.140,208.305,-84.836,173.139,30.474,155.578
C08157=1065.146,208.526,-84.858,173.141,30.478,155.579
C08158=1065.150,208.746,-84.881,173.142,30.481,155.580
C08159=1065.156,208.968,-84.903,173.144,30.485,155.580
C08160=1065.162,209.188,-84.926,173.146,30.488,155.581
C08161=1065.168,209.437,-84.952,173.147,30.493,155.582
C08162=1065.174,209.685,-84.977,173.149,30.496,155.582
C08163=1065.179,209.934,-85.003,173.152,30.501,155.583
C08164=1065.185,210.182,-85.028,173.154,30.504,155.584
C08165=1065.191,210.431,-85.053,173.155,30.509,155.584
C08166=1065.197,210.680,-85.079,173.158,30.513,155.585
C08167=1065.204,210.928,-85.104,173.159,30.517,155.586
C08168=1065.209,211.177,-85.130,173.161,30.521,155.586
C08169=1065.215,211.426,-85.155,173.164,30.525,155.587
C08170=1065.222,211.675,-85.181,173.165,30.529,155.588
C08171=1065.227,211.924,-85.207,173.167,30.533,155.589
C08172=1065.233,212.172,-85.232,173.169,30.537,155.589
C08173=1065.239,212.421,-85.257,173.171,30.542,155.590
C08174=1065.246,212.670,-85.283,173.173,30.545,155.591
C08175=1065.251,212.918,-85.309,173.175,30.550,155.592
C08176=1065.257,213.166,-85.334,173.178,30.553,155.592
C08177=1065.263,213.415,-85.360,173.179,30.558,155.593
C08178=1065.269,213.664,-85.385,173.181,30.562,155.594
C08179=1065.275,213.912,-85.411,173.183,30.566,155.594
C08180=1065.281,214.161,-85.437,173.185,30.570,155.595
C08181=1065.287,214.409,-85.463,173.187,30.574,155.596
C08182=1065.292,214.658,-85.489,173.190,30.578,155.597
C08183=1065.299,214.907,-85.514,173.191,30.582,155.597
C08184=1065.305,215.155,-85.540,173.193,30.586,155.598
C08185=1065.311,215.404,-85.566,173.196,30.590,155.599
C08186=1065.317,215.653,-85.591,173.197,30.594,155.599
C08187=1065.322,215.902,-85.617,173.200,30.599,155.600
C08188=1065.329,216.150,-85.643,173.202,30.602,155.601
C08189=1065.334,216.399,-85.669,173.203,30.607,155.602
C08190=1065.340,216.647,-85.695,173.206,30.611,155.602
C08191=1065.347,216.895,-85.721,173.208,30.615,155.603
C08192=1065.352,217.144,-85.747,173.209,30.619,155.604
C08193=1065.359,217.393,-85.772,173.212,30.623,155.604
C08194=1065.364,217.641,-85.799,173.214,30.627,155.605
C08195=1065.371,217.890,-85.824,173.215,30.631,155.606
C08196=1065.376,218.138,-85.851,173.218,30.635,155.607
C08197=1065.383,218.387,-85.876,173.220,30.639,155.607
C08198=1065.388,218.636,-85.902,173.222,30.643,155.608
C08199=1065.395,218.884,-85.928,173.224,30.647,155.609
C08200=1065.400,219.133,-85.954,173.226,30.651,155.609
C08201=1065.406,219.381,-85.980,173.228,30.655,155.610
C08202=1065.412,219.630,-86.006,173.230,30.659,155.611
C08203=1065.418,219.878,-86.032,173.232,30.663,155.612
C08204=1065.425,220.128,-86.058,173.234,30.667,155.612
C08205=1065.431,220.376,-86.084,173.236,30.671,155.613
C08206=1065.437,220.625,-86.110,173.239,30.675,155.614
C08207=1065.443,220.873,-86.136,173.241,30.679,155.614
C08208=1065.449,221.122,-86.162,173.242,30.683,155.615
C08209=1065.455,221.345,-86.186,173.245,30.687,155.616
C08210=1065.460,221.569,-86.210,173.247,30.690,155.616
C08211=1065.465,221.792,-86.232,173.248,30.694,155.617
C08212=1065.470,222.015,-86.257,173.250,30.698,155.618
C08213=1065.475,222.239,-86.280,173.252,30.702,155.618
C08214=1065.481,222.462,-86.303,173.254,30.705,155.619
C08215=1065.486,222.685,-86.328,173.255,30.708,155.619
C08216=1065.492,222.909,-86.351,173.258,30.712,155.620
C08217=1065.498,223.157,-86.377,173.260,30.717,155.621
C08218=1065.503,223.406,-86.403,173.261,30.720,155.622
C08219=1065.509,223.655,-86.430,173.264,30.724,155.622
C08220=1065.516,223.903,-86.456,173.266,30.729,155.623
C08221=1065.521,224.152,-86.482,173.268,30.732,155.624
C08222=1065.527,224.400,-86.508,173.270,30.737,155.624
C08223=1065.533,224.649,-86.535,173.272,30.740,155.625
C08224=1065.540,224.897,-86.562,173.275,30.745,155.626
C08225=1065.545,225.146,-86.587,173.276,30.749,155.627
C08226=1065.551,225.394,-86.614,173.279,30.753,155.627
C08227=1065.557,225.643,-86.641,173.281,30.757,155.628
C08228=1065.563,225.891,-86.667,173.283,30.761,155.629
C08229=1065.569,226.140,-86.693,173.285,30.765,155.629
C08230=1065.575,226.389,-86.720,173.287,30.769,155.630
C08231=1065.581,226.637,-86.746,173.289,30.773,155.631
C08232=1065.587,226.885,-86.772,173.291,30.777,155.632
C08233=1065.593,227.134,-86.799,173.294,30.781,155.632
C08234=1065.600,227.383,-86.826,173.296,30.784,155.633
C08235=1065.605,227.632,-86.852,173.298,30.789,155.634
C08236=1065.611,227.880,-86.879,173.300,30.793,155.634
C08237=1065.617,228.128,-86.905,173.303,30.797,155.635
C08238=1065.624,228.377,-86.932,173.304,30.801,155.636
C08239=1065.629,228.625,-86.958,173.306,30.805,155.636
C08240=1065.635,228.874,-86.985,173.309,30.808,155.637
C08241=1065.641,229.122,-87.012,173.311,30.813,155.638
C08242=1065.648,229.371,-87.038,173.313,30.817,155.638
C08243=1065.654,229.619,-87.065,173.315,30.820,155.639
C08244=1065.660,229.868,-87.091,173.318,30.825,155.640
C08245=1065.665,230.116,-87.118,173.319,30.828,155.641
C08246=1065.672,230.365,-87.145,173.322,30.833,155.641
C08247=1065.678,230.613,-87.172,173.324,30.837,155.642
C08248=1065.683,230.862,-87.198,173.327,30.840,155.643
C08249=1065.689,231.110,-87.225,173.328,30.845,155.643
C08250=1065.696,231.359,-87.252,173.331,30.849,155.644
C08251=1065.701,231.608,-87.279,173.333,30.853,155.645
C08252=1065.707,231.856,-87.305,173.335,30.857,155.646
C08253=1065.713,232.105,-87.332,173.337,30.860,155.646
C08254=1065.719,232.353,-87.359,173.339,30.865,155.647
C08255=1065.725,232.602,-87.386,173.341,30.869,155.648
C08256=1065.732,232.850,-87.413,173.343,30.872,155.648
C08257=1065.737,233.098,-87.440,173.346,30.877,155.649
C08258=1065.743,233.347,-87.467,173.348,30.881,155.650
C08259=1065.749,233.595,-87.493,173.350,30.884,155.650
C08260=1065.755,233.844,-87.520,173.352,30.889,155.651
C08261=1065.760,234.093,-87.548,173.355,30.893,155.652
C08262=1065.767,234.341,-87.575,173.357,30.897,155.653
C08263=1065.773,234.590,-87.602,173.359,30.901,155.653
C08264=1065.779,234.838,-87.629,173.361,30.904,155.654
C08265=1065.787,235.172,-87.665,173.365,30.910,155.655
C08266=1065.795,235.505,-87.701,173.367,30.916,155.656
C08267=1065.803,235.839,-87.737,173.370,30.921,155.657
C08268=1065.811,236.172,-87.774,173.373,30.926,155.658
C08269=1065.817,236.421,-87.801,173.375,30.930,155.658
C08270=1065.823,236.669,-87.828,173.378,30.934,155.659
C08271=1065.829,236.918,-87.856,173.380,30.938,155.660
C08272=1065.835,237.167,-87.883,173.382,30.942,155.661
C08273=1065.840,237.415,-87.909,173.384,30.946,155.661
C08274=1065.847,237.663,-87.937,173.387,30.950,155.662
C08275=1065.853,237.912,-87.964,173.390,30.954,155.663
C08276=1065.859,238.161,-87.991,173.391,30.958,155.663
C08277=1065.867,238.514,-88.030,173.395,30.963,155.664
C08278=1065.876,238.868,-88.069,173.397,30.969,155.665
C08279=1065.884,239.221,-88.108,173.401,30.975,155.666
C08280=1065.893,239.575,-88.147,173.404,30.980,155.667
C08281=1065.899,239.823,-88.174,173.406,30.985,155.668
C08282=1065.905,240.072,-88.202,173.409,30.989,155.669
C08283=1065.911,240.320,-88.229,173.411,30.992,155.669
C08284=1065.917,240.568,-88.256,173.414,30.997,155.670
C08285=1065.923,240.817,-88.283,173.415,31.000,155.671
C08286=1065.929,241.065,-88.311,173.418,31.004,155.672
C08287=1065.935,241.314,-88.338,173.420,31.009,155.672
C08288=1065.941,241.562,-88.365,173.423,31.012,155.673
C08289=1065.948,241.811,-88.392,173.424,31.016,155.674
C08290=1065.953,242.059,-88.420,173.427,31.020,155.674
C08291=1065.960,242.307,-88.448,173.430,31.024,155.675
C08292=1065.966,242.556,-88.475,173.432,31.028,155.676
C08293=1065.971,242.804,-88.503,173.434,31.032,155.677
C08294=1065.977,243.052,-88.530,173.436,31.036,155.677
C08295=1065.983,243.302,-88.558,173.439,31.040,155.678
C08296=1065.989,243.549,-88.585,173.440,31.044,155.679
C08297=1065.995,243.798,-88.614,173.443,31.048,155.679
C08298=1066.001,244.046,-88.640,173.446,31.052,155.680
C08299=1066.007,244.295,-88.669,173.448,31.056,155.681
C08300=1066.013,244.543,-88.696,173.450,31.060,155.681
C08301=1066.019,244.792,-88.724,173.452,31.064,155.682
C08302=1066.025,245.041,-88.751,173.455,31.068,155.683
C08303=1066.030,245.289,-88.779,173.458,31.072,155.684
C08304=1066.037,245.537,-88.807,173.459,31.076,155.684
C08305=1066.042,245.785,-88.835,173.462,31.080,155.685
C08306=1066.049,246.034,-88.863,173.464,31.084,155.686
C08307=1066.055,246.282,-88.891,173.467,31.088,155.686
C08308=1066.061,246.531,-88.918,173.468,31.092,155.687
C08309=1066.066,246.779,-88.946,173.471,31.096,155.688
C08310=1066.072,247.028,-88.974,173.474,31.100,155.689
C08311=1066.078,247.275,-89.001,173.476,31.104,155.689
C08312=1066.084,247.524,-89.030,173.478,31.108,155.690
C08313=1066.090,247.773,-89.058,173.480,31.112,155.691
C08314=1066.096,248.021,-89.085,173.483,31.116,155.691
C08315=1066.102,248.269,-89.114,173.486,31.120,155.692
C08316=1066.107,248.517,-89.142,173.487,31.124,155.693
C08317=1066.113,248.734,-89.166,173.490,31.128,155.693
C08318=1066.118,248.950,-89.190,173.492,31.131,155.694
C08319=1066.123,249.166,-89.215,173.494,31.135,155.695
C08320=1066.128,249.383,-89.239,173.495,31.138,155.695
C08321=1066.133,249.599,-89.264,173.498,31.141,155.696
C08322=1066.138,249.815,-89.288,173.500,31.145,155.697
C08323=1066.144,250.032,-89.312,173.502,31.149,155.697
C08324=1066.148,250.247,-89.337,173.505,31.152,155.698
C08325=1066.154,250.496,-89.365,173.506,31.156,155.699
C08326=1066.161,250.744,-89.393,173.509,31.160,155.699
C08327=1066.166,250.992,-89.421,173.511,31.164,155.700
C08328=1066.172,251.241,-89.449,173.514,31.168,155.701
C08329=1066.178,251.490,-89.477,173.516,31.172,155.701
C08330=1066.184,251.737,-89.505,173.518,31.176,155.702
C08331=1066.191,251.985,-89.534,173.521,31.180,155.703
C08332=1066.196,252.234,-89.562,173.524,31.184,155.703
C08333=1066.202,252.482,-89.590,173.525,31.188,155.704
C08334=1066.208,252.731,-89.618,173.528,31.192,155.705
C08335=1066.214,252.979,-89.646,173.531,31.196,155.706
C08336=1066.220,253.227,-89.675,173.533,31.200,155.706
C08337=1066.226,253.476,-89.703,173.535,31.204,155.707
C08338=1066.232,253.724,-89.731,173.538,31.208,155.708
C08339=1066.237,253.972,-89.759,173.540,31.212,155.708
C08340=1066.244,254.220,-89.788,173.543,31.216,155.709
C08341=1066.250,254.469,-89.816,173.545,31.220,155.710
C08342=1066.256,254.718,-89.845,173.547,31.224,155.711
C08343=1066.262,254.966,-89.873,173.550,31.228,155.711
C08344=1066.268,255.214,-89.902,173.553,31.232,155.712
C08345=1066.274,255.463,-89.930,173.554,31.236,155.713
C08346=1066.280,255.711,-89.958,173.557,31.240,155.713
C08347=1066.286,255.959,-89.986,173.560,31.244,155.714
C08348=1066.292,256.207,-90.015,173.562,31.248,155.715
C08349=1066.298,256.455,-90.044,173.564,31.252,155.715
C08350=1066.304,256.704,-90.072,173.567,31.255,155.716
C08351=1066.310,256.953,-90.100,173.569,31.260,155.717
C08352=1066.317,257.200,-90.128,173.572,31.263,155.718
C08353=1066.322,257.449,-90.157,173.575,31.267,155.718
C08354=1066.329,257.697,-90.186,173.576,31.272,155.719
C08355=1066.335,257.946,-90.214,173.579,31.275,155.720
C08356=1066.341,258.194,-90.243,173.582,31.279,155.720
C08357=1066.347,258.443,-90.271,173.585,31.284,155.721
C08358=1066.352,258.690,-90.300,173.586,31.287,155.722
C08359=1066.359,258.938,-90.328,173.589,31.291,155.722
C08360=1066.365,259.187,-90.357,173.592,31.295,155.723
C08361=1066.371,259.435,-90.385,173.594,31.299,155.724
C08362=1066.378,259.683,-90.414,173.596,31.303,155.725
C08363=1066.384,259.932,-90.443,173.599,31.307,155.725
C08364=1066.390,260.180,-90.472,173.602,31.311,155.726
C08365=1066.396,260.429,-90.500,173.604,31.315,155.727
C08366=1066.401,260.677,-90.529,173.607,31.319,155.727
C08367=1066.408,260.925,-90.558,173.609,31.322,155.728
C08368=1066.414,261.173,-90.585,173.612,31.327,155.729
C08369=1066.421,261.421,-90.614,173.614,31.330,155.729
C08370=1066.427,261.669,-90.643,173.617,31.334,155.730
C08371=1066.433,261.918,-90.672,173.619,31.338,155.731
C08372=1066.439,262.166,-90.701,173.622,31.342,155.732
C08373=1066.445,262.382,-90.726,173.624,31.346,155.732
C08374=1066.449,262.597,-90.751,173.626,31.349,155.733
C08375=1066.455,262.811,-90.776,173.629,31.352,155.733
C08376=1066.461,263.027,-90.800,173.630,31.356,155.734
C08377=1066.466,263.241,-90.826,173.633,31.359,155.735
C08378=1066.471,263.457,-90.851,173.635,31.362,155.735
C08379=1066.476,263.672,-90.876,173.637,31.366,155.736
C08380=1066.482,263.888,-90.901,173.640,31.369,155.736
C08381=1066.487,264.135,-90.929,173.641,31.374,155.737
C08382=1066.493,264.383,-90.958,173.644,31.377,155.738
C08383=1066.500,264.631,-90.988,173.647,31.381,155.738
C08384=1066.505,264.880,-91.017,173.650,31.386,155.739
C08385=1066.511,265.128,-91.046,173.652,31.389,155.740
C08386=1066.518,265.376,-91.075,173.654,31.394,155.741
C08387=1066.524,265.624,-91.104,173.657,31.397,155.741
C08388=1066.529,265.873,-91.133,173.660,31.401,155.742
C08389=1066.535,266.121,-91.162,173.663,31.406,155.743
C08390=1066.542,266.369,-91.191,173.665,31.409,155.744
C08391=1066.548,266.618,-91.220,173.667,31.414,155.744
C08392=1066.553,266.866,-91.250,173.670,31.417,155.745
C08393=1066.560,267.114,-91.279,173.673,31.421,155.746
C08394=1066.566,267.362,-91.308,173.675,31.425,155.746
C08395=1066.572,267.610,-91.337,173.677,31.429,155.747
C08396=1066.578,267.859,-91.367,173.680,31.434,155.748
C08397=1066.584,268.107,-91.396,173.683,31.437,155.749
C08398=1066.590,268.355,-91.425,173.686,31.441,155.749
C08399=1066.596,268.604,-91.454,173.688,31.445,155.750
C08400=1066.602,268.851,-91.484,173.690,31.449,155.751
C08401=1066.609,269.099,-91.513,173.693,31.454,155.751
C08402=1066.614,269.348,-91.543,173.696,31.457,155.752
C08403=1066.620,269.596,-91.572,173.699,31.461,155.753
C08404=1066.627,269.844,-91.601,173.701,31.465,155.754
C08405=1066.632,270.092,-91.631,173.703,31.469,155.754
C08406=1066.638,270.341,-91.660,173.706,31.474,155.755
C08407=1066.644,270.588,-91.690,173.709,31.477,155.756
C08408=1066.650,270.836,-91.719,173.712,31.482,155.756
C08409=1066.657,271.085,-91.748,173.714,31.485,155.757
C08410=1066.663,271.334,-91.778,173.716,31.489,155.758
C08411=1066.669,271.582,-91.807,173.719,31.493,155.759
C08412=1066.675,271.830,-91.837,173.722,31.497,155.759
C08413=1066.681,272.078,-91.866,173.725,31.502,155.760
C08414=1066.687,272.326,-91.896,173.727,31.505,155.761
C08415=1066.693,272.574,-91.926,173.729,31.510,155.762
C08416=1066.699,272.822,-91.956,173.732,31.513,155.762
C08417=1066.705,273.070,-91.985,173.735,31.517,155.763
C08418=1066.711,273.318,-92.015,173.738,31.522,155.764
C08419=1066.717,273.566,-92.044,173.740,31.525,155.764
C08420=1066.723,273.815,-92.074,173.743,31.530,155.765
C08421=1066.730,274.063,-92.104,173.746,31.533,155.766
C08422=1066.735,274.311,-92.133,173.748,31.538,155.767
C08423=1066.742,274.559,-92.163,173.751,31.541,155.767
C08424=1066.747,274.807,-92.193,173.753,31.546,155.768
C08425=1066.753,275.056,-92.222,173.756,31.550,155.769
C08426=1066.759,275.303,-92.252,173.759,31.554,155.769
C08427=1066.765,275.552,-92.282,173.762,31.558,155.770
C08428=1066.772,275.800,-92.312,173.765,31.562,155.771
C08429=1066.776,276.017,-92.338,173.766,31.566,155.772
C08430=1066.782,276.234,-92.364,173.769,31.569,155.772
C08431=1066.787,276.450,-92.391,173.771,31.573,155.773
C08432=1066.792,276.667,-92.417,173.774,31.576,155.774
C08433=1066.798,276.884,-92.442,173.776,31.579,155.774
C08434=1066.803,277.101,-92.468,173.779,31.583,155.775
C08435=1066.808,277.317,-92.495,173.780,31.587,155.775
C08436=1066.814,277.534,-92.521,173.783,31.590,155.776
C08437=1066.820,277.783,-92.551,173.785,31.594,155.777
C08438=1066.826,278.031,-92.581,173.788,31.598,155.777
C08439=1066.832,278.279,-92.611,173.791,31.602,155.778
C08440=1066.838,278.527,-92.640,173.793,31.606,155.779
C08441=1066.843,278.775,-92.671,173.796,31.610,155.780
C08442=1066.851,279.023,-92.701,173.799,31.614,155.780
C08443=1066.856,279.271,-92.731,173.802,31.619,155.781
C08444=1066.862,279.520,-92.761,173.805,31.622,155.782
C08445=1066.868,279.767,-92.791,173.807,31.627,155.783
C08446=1066.875,280.016,-92.821,173.810,31.630,155.783
C08447=1066.880,280.264,-92.851,173.812,31.635,155.784
C08448=1066.886,280.512,-92.881,173.815,31.638,155.785
C08449=1066.893,280.760,-92.912,173.818,31.643,155.786
C08450=1066.898,281.008,-92.942,173.821,31.647,155.786
C08451=1066.904,281.256,-92.973,173.823,31.651,155.787
C08452=1066.911,281.504,-93.002,173.826,31.655,155.788
C08453=1066.917,281.753,-93.033,173.829,31.659,155.789
C08454=1066.923,282.000,-93.063,173.832,31.663,155.789
C08455=1066.929,282.248,-93.093,173.835,31.668,155.790
C08456=1066.934,282.496,-93.124,173.837,31.671,155.791
C08457=1066.941,282.745,-93.154,173.840,31.676,155.791
C08458=1066.947,282.992,-93.185,173.842,31.680,155.792
C08459=1066.952,283.240,-93.215,173.845,31.684,155.793
C08460=1066.959,283.489,-93.246,173.848,31.688,155.794
C08461=1066.965,283.737,-93.276,173.851,31.692,155.795
C08462=1066.971,283.984,-93.306,173.853,31.696,155.795
C08463=1066.977,284.233,-93.337,173.856,31.700,155.796
C08464=1066.983,284.481,-93.368,173.859,31.704,155.797
C08465=1066.989,284.729,-93.398,173.862,31.708,155.797
C08466=1066.995,284.977,-93.429,173.865,31.713,155.798
C08467=1067.001,285.225,-93.459,173.867,31.716,155.799
C08468=1067.008,285.473,-93.489,173.870,31.721,155.800
C08469=1067.014,285.721,-93.519,173.873,31.725,155.800
C08470=1067.020,285.969,-93.550,173.876,31.729,155.801
C08471=1067.026,286.217,-93.580,173.879,31.733,155.802
C08472=1067.032,286.465,-93.611,173.882,31.737,155.803
C08473=1067.039,286.713,-93.642,173.884,31.741,155.803
C08474=1067.044,286.961,-93.673,173.887,31.745,155.804
C08475=1067.050,287.209,-93.703,173.890,31.749,155.805
C08476=1067.057,287.457,-93.734,173.893,31.754,155.806
C08477=1067.062,287.705,-93.764,173.896,31.757,155.806
C08478=1067.069,287.954,-93.795,173.898,31.762,155.807
C08479=1067.075,288.201,-93.826,173.901,31.766,155.808
C08480=1067.081,288.449,-93.857,173.904,31.770,155.809
C08481=1067.087,288.697,-93.887,173.907,31.774,155.809
C08482=1067.093,288.945,-93.919,173.910,31.778,155.810
C08483=1067.099,289.193,-93.949,173.913,31.782,155.811
C08484=1067.105,289.442,-93.980,173.915,31.786,155.812
C08485=1067.111,289.663,-94.007,173.917,31.790,155.812
C08486=1067.116,289.885,-94.035,173.920,31.794,155.813
C08487=1067.122,290.107,-94.063,173.923,31.798,155.814
C08488=1067.127,290.329,-94.091,173.925,31.801,155.814
C08489=1067.132,290.552,-94.119,173.928,31.805,155.815
C08490=1067.138,290.773,-94.146,173.931,31.809,155.816
C08491=1067.143,290.996,-94.174,173.932,31.812,155.816
C08492=1067.149,291.218,-94.201,173.935,31.816,155.817
C08493=1067.156,291.465,-94.232,173.938,31.820,155.818
C08494=1067.161,291.714,-94.263,173.941,31.825,155.819
C08495=1067.167,291.962,-94.295,173.944,31.828,155.819
C08496=1067.173,292.209,-94.325,173.947,31.833,155.820
C08497=1067.180,292.457,-94.356,173.949,31.837,155.821
C08498=1067.185,292.705,-94.387,173.952,31.841,155.822
C08499=1067.192,292.953,-94.419,173.955,31.845,155.822
C08500=1067.198,293.201,-94.449,173.958,31.849,155.823
C08501=1067.204,293.449,-94.481,173.961,31.854,155.824
C08502=1067.210,293.696,-94.512,173.964,31.858,155.825
C08503=1067.216,293.945,-94.543,173.966,31.862,155.826
C08504=1067.223,294.193,-94.574,173.970,31.866,155.826
C08505=1067.228,294.441,-94.605,173.973,31.870,155.827
C08506=1067.235,294.689,-94.637,173.976,31.875,155.828
C08507=1067.241,294.936,-94.668,173.979,31.879,155.829
C08508=1067.246,295.185,-94.699,173.982,31.883,155.829
C08509=1067.253,295.433,-94.731,173.984,31.887,155.830
C08510=1067.259,295.680,-94.762,173.987,31.891,155.831
C08511=1067.265,295.929,-94.793,173.990,31.896,155.832
C08512=1067.271,296.176,-94.824,173.993,31.900,155.833
C08513=1067.277,296.424,-94.856,173.996,31.904,155.833
C08514=1067.284,296.672,-94.887,173.999,31.908,155.834
C08515=1067.289,296.920,-94.919,174.001,31.912,155.835
C08516=1067.296,297.168,-94.950,174.004,31.917,155.836
C08517=1067.301,297.416,-94.982,174.007,31.921,155.836
C08518=1067.308,297.664,-95.013,174.010,31.925,155.837
C08519=1067.314,297.912,-95.045,174.014,31.930,155.838
C08520=1067.319,298.159,-95.077,174.017,31.934,155.839
C08521=1067.326,298.407,-95.108,174.020,31.938,155.840
C08522=1067.331,298.655,-95.140,174.022,31.942,155.840
C08523=1067.337,298.903,-95.172,174.025,31.947,155.841
C08524=1067.344,299.151,-95.203,174.028,31.951,155.842
C08525=1067.349,299.398,-95.235,174.031,31.955,155.843
C08526=1067.355,299.647,-95.267,174.034,31.959,155.844
C08527=1067.362,299.895,-95.298,174.037,31.964,155.844
C08528=1067.367,300.142,-95.330,174.039,31.968,155.845
C08529=1067.373,300.390,-95.362,174.042,31.972,155.846
C08530=1067.379,300.637,-95.393,174.046,31.977,155.847
C08531=1067.385,300.886,-95.425,174.049,31.981,155.848
C08532=1067.391,301.134,-95.457,174.052,31.985,155.848
C08533=1067.397,301.382,-95.489,174.055,31.990,155.849
C08534=1067.404,301.629,-95.520,174.058,31.994,155.850
C08535=1067.410,301.878,-95.552,174.060,31.999,155.851
C08536=1067.416,302.126,-95.584,174.063,32.003,155.852
C08537=1067.421,302.373,-95.616,174.066,32.007,155.852
C08538=1067.428,302.621,-95.648,174.069,32.011,155.853
C08539=1067.434,302.869,-95.680,174.073,32.016,155.854
C08540=1067.440,303.117,-95.712,174.076,32.020,155.855
C08541=1067.445,303.346,-95.742,174.079,32.024,155.856
C08542=1067.451,303.576,-95.772,174.081,32.028,155.856
C08543=1067.457,303.805,-95.800,174.083,32.032,155.857
C08544=1067.463,304.034,-95.830,174.086,32.036,155.858
C08545=1067.469,304.264,-95.860,174.089,32.040,155.859
C08546=1067.474,304.493,-95.890,174.092,32.044,155.859
C08547=1067.479,304.724,-95.919,174.095,32.048,155.860
C08548=1067.485,304.953,-95.949,174.098,32.052,155.861
C08549=1067.491,305.200,-95.981,174.101,32.056,155.862
C08550=1067.497,305.448,-96.013,174.103,32.060,155.862
C08551=1067.504,305.696,-96.045,174.107,32.065,155.863
C08552=1067.510,305.944,-96.077,174.110,32.070,155.864
C08553=1067.516,306.192,-96.109,174.113,32.074,155.865
C08554=1067.522,306.440,-96.142,174.116,32.078,155.866
C08555=1067.528,306.687,-96.174,174.119,32.082,155.867
C08556=1067.535,306.935,-96.206,174.123,32.087,155.867
C08557=1067.541,307.183,-96.238,174.125,32.091,155.868
C08558=1067.547,307.431,-96.270,174.128,32.095,155.869
C08559=1067.553,307.679,-96.303,174.131,32.100,155.870
C08560=1067.559,307.927,-96.335,174.134,32.104,155.871
C08561=1067.565,308.174,-96.368,174.138,32.109,155.871
C08562=1067.572,308.422,-96.399,174.141,32.113,155.872
C08563=1067.578,308.670,-96.432,174.144,32.117,155.873
C08564=1067.585,308.917,-96.464,174.147,32.122,155.874
C08565=1067.591,309.166,-96.496,174.149,32.126,155.875
C08566=1067.597,309.413,-96.529,174.153,32.130,155.875
C08567=1067.603,309.661,-96.561,174.156,32.135,155.876
C08568=1067.609,309.909,-96.594,174.159,32.139,155.877
C08569=1067.616,310.156,-96.626,174.162,32.144,155.878
C08570=1067.622,310.405,-96.658,174.166,32.148,155.879
C08571=1067.628,310.652,-96.691,174.169,32.152,155.880
C08572=1067.635,310.900,-96.724,174.172,32.156,155.880
C08573=1067.641,311.148,-96.756,174.174,32.161,155.881
C08574=1067.647,311.396,-96.788,174.177,32.166,155.882
C08575=1067.653,311.643,-96.821,174.181,32.170,155.883
C08576=1067.659,311.891,-96.853,174.184,32.174,155.884
C08577=1067.666,312.139,-96.886,174.187,32.178,155.885
C08578=1067.673,312.386,-96.918,174.190,32.183,155.885
C08579=1067.679,312.634,-96.951,174.194,32.187,155.886
C08580=1067.685,312.881,-96.984,174.197,32.192,155.887
C08581=1067.691,313.130,-97.016,174.199,32.196,155.888
C08582=1067.697,313.377,-97.048,174.203,32.200,155.889
C08583=1067.704,313.626,-97.081,174.206,32.205,155.889
C08584=1067.711,313.873,-97.114,174.209,32.209,155.890
C08585=1067.717,314.121,-97.147,174.212,32.214,155.891
C08586=1067.723,314.368,-97.180,174.216,32.218,155.892
C08587=1067.729,314.616,-97.213,174.219,32.223,155.893
C08588=1067.735,314.864,-97.246,174.222,32.227,155.894
C08589=1067.741,315.111,-97.278,174.224,32.232,155.895
C08590=1067.747,315.359,-97.312,174.228,32.236,155.895
C08591=1067.753,315.607,-97.345,174.231,32.241,155.896
C08592=1067.759,315.855,-97.378,174.234,32.245,155.897
C08593=1067.765,316.102,-97.411,174.237,32.250,155.898
C08594=1067.771,316.350,-97.443,174.241,32.254,155.899
C08595=1067.777,316.598,-97.477,174.244,32.259,155.900
C08596=1067.783,316.845,-97.509,174.247,32.264,155.901
C08597=1067.790,317.077,-97.541,174.250,32.268,155.902
C08598=1067.795,317.308,-97.572,174.252,32.272,155.902
C08599=1067.801,317.540,-97.603,174.255,32.277,155.903
C08600=1067.806,317.771,-97.633,174.258,32.281,155.904
C08601=1067.812,318.002,-97.664,174.262,32.285,155.905
C08602=1067.818,318.234,-97.696,174.265,32.289,155.906
C08603=1067.823,318.464,-97.727,174.268,32.294,155.906
C08604=1067.829,318.697,-97.757,174.271,32.298,155.907
C08605=1067.835,318.944,-97.791,174.274,32.303,155.908
C08606=1067.841,319.191,-97.824,174.277,32.307,155.909
C08607=1067.848,319.439,-97.857,174.281,32.312,155.910
C08608=1067.853,319.687,-97.890,174.283,32.317,155.911
C08609=1067.860,319.935,-97.924,174.286,32.321,155.912
C08610=1067.866,320.183,-97.957,174.290,32.326,155.913
C08611=1067.872,320.430,-97.990,174.293,32.331,155.913
C08612=1067.878,320.677,-98.024,174.296,32.335,155.914
C08613=1067.884,320.925,-98.057,174.300,32.340,155.915
C08614=1067.891,321.173,-98.091,174.303,32.344,155.916
C08615=1067.897,321.421,-98.124,174.306,32.349,155.917
C08616=1067.903,321.668,-98.158,174.310,32.354,155.918
C08617=1067.910,321.916,-98.191,174.313,32.358,155.919
C08618=1067.915,322.164,-98.225,174.316,32.363,155.920
C08619=1067.922,322.411,-98.258,174.319,32.367,155.921
C08620=1067.928,322.659,-98.291,174.322,32.372,155.921
C08621=1067.935,322.907,-98.325,174.325,32.377,155.922
C08622=1067.940,323.154,-98.359,174.329,32.381,155.923
C08623=1067.947,323.401,-98.392,174.332,32.386,155.924
C08624=1067.953,323.650,-98.426,174.336,32.391,155.925
C08625=1067.960,323.897,-98.459,174.339,32.395,155.926
C08626=1067.966,324.146,-98.493,174.342,32.400,155.927
C08627=1067.972,324.393,-98.527,174.346,32.405,155.928
C08628=1067.978,324.640,-98.560,174.349,32.410,155.929
C08629=1067.985,324.889,-98.594,174.351,32.414,155.930
C08630=1067.991,325.135,-98.628,174.355,32.419,155.930
C08631=1067.998,325.383,-98.662,174.358,32.423,155.931
C08632=1068.004,325.631,-98.695,174.362,32.428,155.932
C08633=1068.010,325.878,-98.729,174.365,32.433,155.933
C08634=1068.016,326.126,-98.763,174.368,32.437,155.934
C08635=1068.022,326.374,-98.796,174.372,32.442,155.935
C08636=1068.029,326.622,-98.830,174.375,32.447,155.936
C08637=1068.036,326.869,-98.864,174.379,32.452,155.937
C08638=1068.042,327.117,-98.898,174.382,32.456,155.938
C08639=1068.049,327.364,-98.932,174.386,32.461,155.939
C08640=1068.055,327.612,-98.965,174.389,32.466,155.939
C08641=1068.061,327.860,-99.000,174.392,32.470,155.940
C08642=1068.068,328.107,-99.033,174.395,32.475,155.941
C08643=1068.074,328.355,-99.067,174.398,32.480,155.942
C08644=1068.080,328.603,-99.102,174.402,32.485,155.943
C08645=1068.087,328.850,-99.135,174.405,32.489,155.944
C08646=1068.093,329.098,-99.170,174.409,32.494,155.945
C08647=1068.100,329.346,-99.203,174.412,32.499,155.946
C08648=1068.106,329.593,-99.237,174.416,32.503,155.947
C08649=1068.112,329.841,-99.271,174.419,32.508,155.948
C08650=1068.119,330.088,-99.305,174.422,32.513,155.949
C08651=1068.125,330.336,-99.339,174.426,32.518,155.950
C08652=1068.132,330.584,-99.374,174.429,32.523,155.951
C08653=1068.138,330.812,-99.405,174.433,32.527,155.951
C08654=1068.145,331.040,-99.437,174.436,32.532,155.952
C08655=1068.150,331.268,-99.468,174.438,32.536,155.953
C08656=1068.155,331.497,-99.500,174.441,32.540,155.954
C08657=1068.161,331.725,-99.531,174.444,32.545,155.955
C08658=1068.167,331.953,-99.563,174.448,32.550,155.956
C08659=1068.172,332.181,-99.595,174.451,32.554,155.957
C08660=1068.179,332.409,-99.626,174.454,32.558,155.958
C08661=1068.185,332.657,-99.661,174.458,32.563,155.958
C08662=1068.191,332.905,-99.695,174.461,32.569,155.959
C08663=1068.198,333.153,-99.729,174.464,32.573,155.960
C08664=1068.204,333.399,-99.764,174.468,32.578,155.961
C08665=1068.210,333.647,-99.799,174.471,32.583,155.962
C08666=1068.217,333.895,-99.833,174.475,32.588,155.963
C08667=1068.223,334.142,-99.868,174.478,32.593,155.964
C08668=1068.229,334.390,-99.902,174.482,32.598,155.965
C08669=1068.236,334.638,-99.937,174.486,32.603,155.966
C08670=1068.242,334.885,-99.971,174.489,32.608,155.967
C08671=1068.249,335.133,-100.006,174.493,32.613,155.968
C08672=1068.255,335.381,-100.040,174.495,32.618,155.969
C08673=1068.261,335.627,-100.075,174.499,32.623,155.970
C08674=1068.267,335.876,-100.110,174.502,32.628,155.971
C08675=1068.274,336.123,-100.145,174.506,32.632,155.972
C08676=1068.279,336.370,-100.179,174.509,32.638,155.973
C08677=1068.286,336.618,-100.214,174.513,32.643,155.974
C08678=1068.293,336.866,-100.249,174.516,32.647,155.975
C08679=1068.299,337.113,-100.284,174.520,32.653,155.976
C08680=1068.305,337.360,-100.318,174.523,32.657,155.977
C08681=1068.312,337.608,-100.353,174.527,32.663,155.978
C08682=1068.319,337.856,-100.387,174.531,32.668,155.979
C08683=1068.325,338.103,-100.423,174.534,32.673,155.980
C08684=1068.331,338.350,-100.458,174.538,32.678,155.981
C08685=1068.337,338.598,-100.492,174.541,32.683,155.982
C08686=1068.344,338.845,-100.527,174.545,32.688,155.983
C08687=1068.350,339.093,-100.563,174.548,32.693,155.984
C08688=1068.356,339.340,-100.597,174.552,32.698,155.985
C08689=1068.363,339.588,-100.632,174.555,32.703,155.986
C08690=1068.369,339.835,-100.668,174.559,32.708,155.987
C08691=1068.375,340.083,-100.703,174.563,32.713,155.988
C08692=1068.382,340.331,-100.738,174.566,32.719,155.989
C08693=1068.389,340.578,-100.773,174.570,32.724,155.990
C08694=1068.394,340.825,-100.808,174.573,32.729,155.991
C08695=1068.401,341.072,-100.843,174.576,32.734,155.992
C08696=1068.408,341.320,-100.878,174.580,32.739,155.993
C08697=1068.414,341.567,-100.914,174.583,32.744,155.994
C08698=1068.420,341.815,-100.949,174.587,32.749,155.995
C08699=1068.427,342.063,-100.984,174.591,32.755,155.996
C08700=1068.433,342.310,-101.019,174.594,32.759,155.997
C08701=1068.439,342.557,-101.054,174.598,32.765,155.998
C08702=1068.446,342.804,-101.089,174.601,32.770,155.999
C08703=1068.452,343.052,-101.125,174.605,32.775,156.000
C08704=1068.459,343.299,-101.160,174.609,32.781,156.001
C08705=1068.465,343.547,-101.195,174.612,32.785,156.002
C08706=1068.471,343.794,-101.231,174.616,32.791,156.003
C08707=1068.478,344.042,-101.266,174.620,32.796,156.005
C08708=1068.484,344.290,-101.302,174.623,32.801,156.006
C08709=1068.490,344.515,-101.335,174.627,32.806,156.007
C08710=1068.496,344.741,-101.367,174.630,32.811,156.007
C08711=1068.502,344.966,-101.399,174.633,32.816,156.008
C08712=1068.508,345.192,-101.432,174.637,32.821,156.009
C08713=1068.514,345.418,-101.464,174.640,32.826,156.010
C08714=1068.520,345.644,-101.496,174.643,32.830,156.011
C08715=1068.525,345.870,-101.530,174.647,32.835,156.012
C08716=1068.531,346.096,-101.562,174.650,32.840,156.013
C08717=1068.538,346.343,-101.597,174.654,32.845,156.014
C08718=1068.544,346.590,-101.633,174.657,32.851,156.016
C08719=1068.551,346.838,-101.669,174.661,32.856,156.017
C08720=1068.557,347.085,-101.704,174.665,32.862,156.018
C08721=1068.564,347.332,-101.741,174.668,32.867,156.019
C08722=1068.570,347.580,-101.776,174.672,32.872,156.020
C08723=1068.576,347.827,-101.811,174.676,32.877,156.021
C08724=1068.583,348.074,-101.848,174.680,32.883,156.022
C08725=1068.590,348.322,-101.883,174.683,32.888,156.023
C08726=1068.596,348.569,-101.919,174.687,32.894,156.024
C08727=1068.602,348.816,-101.955,174.691,32.899,156.025
C08728=1068.609,349.064,-101.990,174.694,32.904,156.026
C08729=1068.615,349.311,-102.027,174.698,32.910,156.027
C08730=1068.622,349.559,-102.063,174.702,32.915,156.028
C08731=1068.629,349.806,-102.099,174.706,32.921,156.030
C08732=1068.635,350.054,-102.134,174.709,32.926,156.031
C08733=1068.641,350.301,-102.171,174.713,32.931,156.032
C08734=1068.648,350.547,-102.207,174.717,32.937,156.033
C08735=1068.654,350.795,-102.243,174.721,32.943,156.034
C08736=1068.661,351.042,-102.279,174.724,32.948,156.035
C08737=1068.667,351.290,-102.316,174.728,32.953,156.036
C08738=1068.674,351.537,-102.351,174.732,32.959,156.037
C08739=1068.681,351.784,-102.387,174.736,32.964,156.038
C08740=1068.687,352.031,-102.424,174.739,32.970,156.040
C08741=1068.693,352.279,-102.460,174.743,32.975,156.041
C08742=1068.699,352.526,-102.496,174.747,32.981,156.042
C08743=1068.707,352.773,-102.532,174.751,32.986,156.043
C08744=1068.713,353.021,-102.569,174.754,32.992,156.044
C08745=1068.719,353.268,-102.604,174.758,32.998,156.045
C08746=1068.726,353.515,-102.641,174.762,33.003,156.046
C08747=1068.732,353.762,-102.677,174.766,33.009,156.047
C08748=1068.739,354.010,-102.714,174.770,33.015,156.049
C08749=1068.745,354.257,-102.751,174.773,33.020,156.050
C08750=1068.752,354.504,-102.787,174.777,33.026,156.051
C08751=1068.758,354.751,-102.823,174.781,33.031,156.052
C08752=1068.765,354.999,-102.860,174.785,33.037,156.053
C08753=1068.771,355.246,-102.897,174.789,33.043,156.054
C08754=1068.778,355.493,-102.933,174.793,33.048,156.056
C08755=1068.784,355.740,-102.970,174.797,33.054,156.057
C08756=1068.791,355.988,-103.006,174.801,33.060,156.058
C08757=1068.797,356.235,-103.043,174.805,33.065,156.059
C08758=1068.803,356.482,-103.079,174.809,33.071,156.060
C08759=1068.810,356.730,-103.116,174.813,33.077,156.061
C08760=1068.817,356.977,-103.152,174.816,33.083,156.063
C08761=1068.823,357.224,-103.189,174.820,33.088,156.064
C08762=1068.830,357.471,-103.226,174.824,33.094,156.065
C08763=1068.837,357.718,-103.263,174.828,33.100,156.066
C08764=1068.843,357.965,-103.299,174.832,33.105,156.067
C08765=1068.850,358.193,-103.333,174.835,33.111,156.068
C08766=1068.856,358.421,-103.367,174.839,33.116,156.069
C08767=1068.862,358.648,-103.401,174.842,33.121,156.071
C08768=1068.868,358.876,-103.435,174.846,33.127,156.072
C08769=1068.874,359.104,-103.468,174.850,33.132,156.073
C08770=1068.880,359.331,-103.503,174.853,33.137,156.074
C08771=1068.886,359.559,-103.537,174.857,33.143,156.075
C08772=1068.893,359.787,-103.571,174.860,33.148,156.076
C08773=1068.898,360.034,-103.608,174.864,33.154,156.077
C08774=1068.905,360.281,-103.645,174.868,33.160,156.079
C08775=1068.912,360.528,-103.682,174.873,33.166,156.080
C08776=1068.918,360.775,-103.719,174.877,33.172,156.081
C08777=1068.926,361.022,-103.756,174.881,33.177,156.082
C08778=1068.931,361.270,-103.793,174.885,33.184,156.084
C08779=1068.938,361.517,-103.831,174.889,33.189,156.085
C08780=1068.945,361.764,-103.867,174.893,33.195,156.086
C08781=1068.952,362.011,-103.905,174.896,33.201,156.087
C08782=1068.958,362.258,-103.941,174.900,33.207,156.088
C08783=1068.965,362.505,-103.979,174.904,33.213,156.090
C08784=1068.971,362.753,-104.016,174.908,33.219,156.091
C08785=1068.978,363.000,-104.053,174.912,33.225,156.092
C08786=1068.985,363.246,-104.091,174.916,33.231,156.093
C08787=1068.992,363.494,-104.129,174.920,33.237,156.095
C08788=1068.998,363.741,-104.165,174.924,33.243,156.096
C08789=1069.005,363.988,-104.203,174.929,33.249,156.097
C08790=1069.012,364.235,-104.241,174.933,33.255,156.098
C08791=1069.018,364.482,-104.277,174.937,33.261,156.100
C08792=1069.025,364.729,-104.315,174.941,33.267,156.101
C08793=1069.031,364.976,-104.352,174.945,33.273,156.102
C08794=1069.038,365.223,-104.390,174.949,33.280,156.103
C08795=1069.044,365.470,-104.428,174.953,33.285,156.105
C08796=1069.052,365.717,-104.465,174.957,33.292,156.106
C08797=1069.058,365.965,-104.503,174.961,33.298,156.107
C08798=1069.065,366.211,-104.541,174.965,33.304,156.109
C08799=1069.071,366.458,-104.579,174.970,33.310,156.110
C08800=1069.077,366.705,-104.616,174.974,33.316,156.111
C08801=1069.084,366.952,-104.654,174.978,33.323,156.113
C08802=1069.091,367.200,-104.692,174.982,33.329,156.114
C08803=1069.098,367.446,-104.729,174.986,33.335,156.115
C08804=1069.104,367.694,-104.767,174.990,33.341,156.116
C08805=1069.111,367.941,-104.805,174.994,33.347,156.118
C08806=1069.117,368.188,-104.843,174.998,33.354,156.119
C08807=1069.124,368.435,-104.880,175.002,33.360,156.120
C08808=1069.131,368.682,-104.918,175.007,33.366,156.122
C08809=1069.138,368.928,-104.956,175.011,33.373,156.123
C08810=1069.144,369.175,-104.994,175.015,33.379,156.124
C08811=1069.151,369.423,-105.032,175.019,33.385,156.126
C08812=1069.158,369.670,-105.070,175.023,33.392,156.127
C08813=1069.164,369.916,-105.108,175.027,33.398,156.128
C08814=1069.172,370.163,-105.146,175.031,33.404,156.130
C08815=1069.178,370.411,-105.184,175.035,33.410,156.131
C08816=1069.185,370.657,-105.223,175.040,33.417,156.132
C08817=1069.192,370.904,-105.260,175.044,33.423,156.134
C08818=1069.198,371.151,-105.298,175.048,33.429,156.135
C08819=1069.206,371.398,-105.336,175.052,33.436,156.136
C08820=1069.212,371.645,-105.375,175.057,33.443,156.138
C08821=1069.218,371.881,-105.411,175.060,33.448,156.139
C08822=1069.225,372.118,-105.448,175.064,33.454,156.140
C08823=1069.232,372.353,-105.484,175.069,33.461,156.142
C08824=1069.238,372.590,-105.521,175.073,33.467,156.143
C08825=1069.244,372.826,-105.558,175.077,33.473,156.144
C08826=1069.252,373.063,-105.594,175.081,33.479,156.146
C08827=1069.258,373.299,-105.631,175.085,33.485,156.147
C08828=1069.264,373.535,-105.668,175.089,33.492,156.148
C08829=1069.272,373.782,-105.706,175.093,33.498,156.150
C08830=1069.278,374.029,-105.744,175.098,33.505,156.151
C08831=1069.284,374.275,-105.783,175.102,33.512,156.153
C08832=1069.291,374.522,-105.822,175.106,33.518,156.154
C08833=1069.298,374.769,-105.861,175.111,33.525,156.155
C08834=1069.304,375.017,-105.899,175.115,33.531,156.157
C08835=1069.311,375.263,-105.938,175.119,33.538,156.158
C08836=1069.318,375.510,-105.976,175.124,33.545,156.160
C08837=1069.325,375.757,-106.015,175.128,33.551,156.161
C08838=1069.332,376.004,-106.054,175.132,33.558,156.163
C08839=1069.339,376.251,-106.093,175.136,33.564,156.164
C08840=1069.345,376.497,-106.132,175.141,33.571,156.165
C08841=1069.352,376.745,-106.170,175.146,33.578,156.167
C08842=1069.359,376.992,-106.209,175.150,33.585,156.168
C08843=1069.365,377.239,-106.248,175.154,33.592,156.170
C08844=1069.373,377.485,-106.286,175.158,33.598,156.171
C08845=1069.380,377.732,-106.325,175.163,33.605,156.173
C08846=1069.387,377.978,-106.364,175.168,33.612,156.174
C08847=1069.394,378.225,-106.403,175.172,33.619,156.176
C08848=1069.401,378.472,-106.442,175.176,33.626,156.177
C08849=1069.407,378.719,-106.481,175.180,33.632,156.179
C08850=1069.414,378.965,-106.520,175.185,33.639,156.180
C08851=1069.421,379.212,-106.558,175.190,33.646,156.182
C08852=1069.428,379.459,-106.597,175.194,33.653,156.183
C08853=1069.435,379.705,-106.637,175.198,33.660,156.184
C08854=1069.442,379.952,-106.676,175.203,33.667,156.186
C08855=1069.449,380.200,-106.715,175.207,33.673,156.187
C08856=1069.456,380.446,-106.754,175.212,33.681,156.189
C08857=1069.463,380.693,-106.793,175.216,33.687,156.191
C08858=1069.469,380.940,-106.833,175.221,33.694,156.192
C08859=1069.476,381.187,-106.871,175.225,33.701,156.193
C08860=1069.484,381.434,-106.911,175.230,33.708,156.195
C08861=1069.491,381.680,-106.950,175.234,33.715,156.197
C08862=1069.498,381.927,-106.990,175.239,33.722,156.198
C08863=1069.504,382.174,-107.029,175.243,33.729,156.200
C08864=1069.511,382.420,-107.069,175.247,33.736,156.201
C08865=1069.518,382.667,-107.108,175.253,33.744,156.203
C08866=1069.525,382.913,-107.147,175.257,33.751,156.204
C08867=1069.531,383.161,-107.187,175.261,33.758,156.206
C08868=1069.539,383.407,-107.227,175.266,33.765,156.207
C08869=1069.546,383.653,-107.266,175.271,33.772,156.209
C08870=1069.552,383.900,-107.306,175.275,33.779,156.211
C08871=1069.559,384.147,-107.345,175.279,33.787,156.212
C08872=1069.566,384.394,-107.386,175.285,33.794,156.214
C08873=1069.573,384.641,-107.424,175.289,33.801,156.215
C08874=1069.580,384.887,-107.464,175.293,33.808,156.217
C08875=1069.587,385.134,-107.504,175.298,33.815,156.218
C08876=1069.594,385.380,-107.544,175.303,33.823,156.220
C08877=1069.601,385.636,-107.585,175.308,33.830,156.222
C08878=1069.608,385.892,-107.626,175.312,33.838,156.223
C08879=1069.615,386.147,-107.668,175.318,33.846,156.225
C08880=1069.623,386.403,-107.709,175.322,33.853,156.227
C08881=1069.630,386.649,-107.749,175.327,33.861,156.228
C08882=1069.637,386.896,-107.788,175.331,33.868,156.230
C08883=1069.644,387.143,-107.829,175.336,33.875,156.232
C08884=1069.651,387.389,-107.868,175.341,33.883,156.233
C08885=1069.658,387.635,-107.908,175.345,33.890,156.235
C08886=1069.665,387.883,-107.948,175.351,33.897,156.236
C08887=1069.672,388.129,-107.988,175.355,33.905,156.238
C08888=1069.679,388.376,-108.028,175.359,33.912,156.240
C08889=1069.686,388.622,-108.068,175.365,33.919,156.241
C08890=1069.694,388.869,-108.109,175.369,33.927,156.243
C08891=1069.701,389.115,-108.149,175.374,33.935,156.245
C08892=1069.708,389.362,-108.189,175.378,33.942,156.246
C08893=1069.715,389.608,-108.229,175.384,33.950,156.248
C08894=1069.723,389.855,-108.270,175.388,33.957,156.250
C08895=1069.729,390.101,-108.310,175.393,33.965,156.251
C08896=1069.737,390.348,-108.350,175.398,33.973,156.253
C08897=1069.743,390.595,-108.390,175.403,33.980,156.255
C08898=1069.751,390.841,-108.430,175.407,33.988,156.257
C08899=1069.758,391.088,-108.471,175.413,33.995,156.258
C08900=1069.765,391.334,-108.512,175.417,34.003,156.260
C08901=1069.773,391.581,-108.552,175.423,34.010,156.262
C08902=1069.779,391.827,-108.593,175.427,34.018,156.263
C08903=1069.786,392.074,-108.633,175.432,34.026,156.265
C08904=1069.794,392.320,-108.673,175.437,34.034,156.267
C08905=1069.801,392.567,-108.714,175.442,34.042,156.269
C08906=1069.808,392.813,-108.755,175.446,34.049,156.270
C08907=1069.814,393.060,-108.795,175.452,34.057,156.272
C08908=1069.822,393.306,-108.836,175.456,34.065,156.274
C08909=1069.830,393.553,-108.877,175.462,34.073,156.276
C08910=1069.836,393.799,-108.917,175.466,34.081,156.277
C08911=1069.843,394.046,-108.958,175.471,34.089,156.279
C08912=1069.851,394.292,-108.999,175.476,34.097,156.281
C08913=1069.858,394.538,-109.040,175.481,34.105,156.283
C08914=1069.865,394.785,-109.080,175.485,34.113,156.285
C08915=1069.872,395.032,-109.122,175.491,34.121,156.286
C08916=1069.880,395.278,-109.163,175.496,34.129,156.288
C08917=1069.886,395.524,-109.204,175.501,34.137,156.290
C08918=1069.894,395.771,-109.245,175.506,34.145,156.292
C08919=1069.901,396.018,-109.286,175.511,34.153,156.294
C08920=1069.909,396.264,-109.327,175.516,34.161,156.295
C08921=1069.916,396.510,-109.368,175.521,34.169,156.297
C08922=1069.923,396.756,-109.409,175.526,34.177,156.299
C08923=1069.930,397.003,-109.450,175.531,34.185,156.301
C08924=1069.938,397.249,-109.491,175.536,34.193,156.303
C08925=1069.945,397.496,-109.533,175.541,34.202,156.305
C08926=1069.952,397.743,-109.574,175.547,34.210,156.306
C08927=1069.959,397.989,-109.615,175.551,34.218,156.308
C08928=1069.967,398.236,-109.656,175.556,34.227,156.310
C08929=1069.974,398.482,-109.698,175.562,34.235,156.312
C08930=1069.981,398.728,-109.739,175.566,34.243,156.314
C08931=1069.988,398.974,-109.780,175.572,34.251,156.316
C08932=1069.995,399.221,-109.822,175.577,34.260,156.318
C08933=1070.003,399.493,-109.868,175.583,34.269,156.320
C08934=1070.011,399.764,-109.914,175.588,34.278,156.322
C08935=1070.019,400.036,-109.960,175.594,34.287,156.324
C08936=1070.028,400.307,-110.006,175.599,34.297,156.326
C08937=1070.035,400.554,-110.047,175.605,34.305,156.328
C08938=1070.042,400.800,-110.089,175.610,34.314,156.330
C08939=1070.050,401.046,-110.130,175.615,34.322,156.332
C08940=1070.057,401.292,-110.172,175.620,34.331,156.334
C08941=1070.065,401.539,-110.213,175.626,34.339,156.336
C08942=1070.071,401.785,-110.256,175.631,34.348,156.338
C08943=1070.079,402.032,-110.297,175.636,34.356,156.340
C08944=1070.086,402.278,-110.339,175.642,34.365,156.342
C08945=1070.094,402.524,-110.381,175.647,34.373,156.344
C08946=1070.101,402.770,-110.422,175.653,34.382,156.346
C08947=1070.109,403.017,-110.465,175.657,34.391,156.348
C08948=1070.116,403.263,-110.507,175.663,34.400,156.350
C08949=1070.124,403.509,-110.549,175.668,34.408,156.352
C08950=1070.130,403.756,-110.591,175.674,34.417,156.354
C08951=1070.138,404.002,-110.633,175.679,34.426,156.356
C08952=1070.146,404.248,-110.675,175.684,34.435,156.358
C08953=1070.153,404.495,-110.718,175.689,34.444,156.360
C08954=1070.161,404.741,-110.760,175.695,34.452,156.362
C08955=1070.168,404.987,-110.802,175.701,34.461,156.364
C08956=1070.175,405.233,-110.844,175.706,34.470,156.366
C08957=1070.183,405.480,-110.887,175.712,34.479,156.368
C08958=1070.190,405.726,-110.929,175.717,34.488,156.370
C08959=1070.198,405.972,-110.971,175.722,34.497,156.372
C08960=1070.205,406.219,-111.014,175.728,34.506,156.374
C08961=1070.213,406.465,-111.056,175.733,34.515,156.376
C08962=1070.220,406.712,-111.098,175.739,34.524,156.379
C08963=1070.227,406.958,-111.140,175.744,34.533,156.381
C08964=1070.235,407.204,-111.184,175.750,34.542,156.383
C08965=1070.242,407.450,-111.226,175.756,34.552,156.385
C08966=1070.249,407.696,-111.268,175.761,34.561,156.387
C08967=1070.257,407.943,-111.312,175.767,34.570,156.389
C08968=1070.264,408.189,-111.355,175.773,34.579,156.391
C08969=1070.272,408.436,-111.397,175.778,34.589,156.394
C08970=1070.279,408.681,-111.440,175.784,34.598,156.396
C08971=1070.286,408.928,-111.483,175.790,34.607,156.398
C08972=1070.295,409.174,-111.526,175.795,34.616,156.400
C08973=1070.302,409.420,-111.568,175.801,34.626,156.402
C08974=1070.309,409.666,-111.612,175.807,34.635,156.404
C08975=1070.317,409.912,-111.654,175.812,34.645,156.407
C08976=1070.325,410.159,-111.697,175.818,34.654,156.409
C08977=1070.332,410.405,-111.740,175.824,34.663,156.411
C08978=1070.340,410.651,-111.783,175.829,34.673,156.413
C08979=1070.347,410.897,-111.826,175.835,34.682,156.415
C08980=1070.355,411.144,-111.869,175.841,34.692,156.418
C08981=1070.363,411.390,-111.912,175.847,34.701,156.420
C08982=1070.370,411.635,-111.955,175.852,34.711,156.422
C08983=1070.378,411.882,-111.999,175.858,34.720,156.424
C08984=1070.385,412.127,-112.042,175.864,34.730,156.427
C08985=1070.394,412.374,-112.085,175.869,34.739,156.429
C08986=1070.401,412.620,-112.128,175.875,34.749,156.431
C08987=1070.408,412.866,-112.172,175.881,34.759,156.433
C08988=1070.416,413.112,-112.215,175.888,34.769,156.436
C08989=1070.430,413.527,-112.288,175.897,34.785,156.440
C08990=1070.443,413.942,-112.361,175.907,34.802,156.444
C08991=1070.456,414.356,-112.435,175.918,34.818,156.448
C08992=1070.469,414.771,-112.508,175.928,34.834,156.451
C08993=1070.477,415.018,-112.552,175.934,34.845,156.454
C08994=1070.485,415.264,-112.596,175.940,34.854,156.456
C08995=1070.492,415.509,-112.639,175.945,34.865,156.459
C08996=1070.500,415.755,-112.683,175.951,34.875,156.461
C08997=1070.508,416.002,-112.727,175.958,34.885,156.463
C08998=1070.516,416.248,-112.771,175.964,34.895,156.466
C08999=1070.524,416.494,-112.815,175.970,34.905,156.468
C09000=1070.531,416.739,-112.859,175.976,34.915,156.471
C09001=1070.539,416.985,-112.902,175.983,34.925,156.473
C09002=1070.547,417.231,-112.947,175.988,34.936,156.475
C09003=1070.554,417.478,-112.991,175.994,34.946,156.478
C09004=1070.562,417.724,-113.035,176.001,34.956,156.480
C09005=1070.570,417.969,-113.079,176.007,34.966,156.483
C09006=1070.578,418.216,-113.123,176.013,34.977,156.485
C09007=1070.586,418.461,-113.167,176.020,34.987,156.488
C09008=1070.594,418.707,-113.212,176.026,34.997,156.490
C09009=1070.602,418.953,-113.255,176.032,35.008,156.493
C09010=1070.610,419.199,-113.300,176.039,35.018,156.495
C09011=1070.617,419.445,-113.345,176.045,35.029,156.498
C09012=1070.625,419.691,-113.389,176.052,35.040,156.500
C09013=1070.633,419.937,-113.433,176.058,35.050,156.503
C09014=1070.641,420.183,-113.478,176.065,35.060,156.505
C09015=1070.649,420.428,-113.522,176.071,35.071,156.508
C09016=1070.657,420.674,-113.566,176.077,35.082,156.511
C09017=1070.665,420.920,-113.611,176.083,35.092,156.513
C09018=1070.673,421.167,-113.656,176.089,35.103,156.516
C09019=1070.682,421.412,-113.700,176.097,35.114,156.518
C09020=1070.689,421.658,-113.745,176.103,35.125,156.521
C09021=1070.697,421.904,-113.790,176.110,35.135,156.523
C09022=1070.705,422.150,-113.834,176.116,35.146,156.526
C09023=1070.713,422.395,-113.880,176.123,35.157,156.529
C09024=1070.721,422.641,-113.924,176.129,35.168,156.531
C09025=1070.729,422.888,-113.969,176.136,35.179,156.534
C09026=1070.737,423.133,-114.014,176.143,35.190,156.537
C09027=1070.744,423.379,-114.059,176.149,35.201,156.539
C09028=1070.753,423.624,-114.104,176.156,35.212,156.542
C09029=1070.765,423.977,-114.169,176.165,35.228,156.546
C09030=1070.776,424.329,-114.233,176.175,35.244,156.550
C09031=1070.788,424.681,-114.298,176.185,35.260,156.554
C09032=1070.800,425.033,-114.363,176.194,35.276,156.558
C09033=1070.807,425.279,-114.408,176.201,35.287,156.560
C09034=1070.816,425.524,-114.453,176.208,35.298,156.563
C09035=1070.824,425.771,-114.499,176.215,35.310,156.566
C09036=1070.832,426.016,-114.544,176.222,35.321,156.569
C09037=1070.840,426.262,-114.590,176.228,35.332,156.572
C09038=1070.849,426.507,-114.635,176.235,35.343,156.574
C09039=1070.857,426.753,-114.681,176.242,35.355,156.577
C09040=1070.865,426.999,-114.726,176.250,35.367,156.580
C09041=1070.875,427.293,-114.780,176.257,35.380,156.583
C09042=1070.885,427.587,-114.836,176.266,35.394,156.587
C09043=1070.894,427.881,-114.891,176.274,35.408,156.590
C09044=1070.904,428.175,-114.945,176.283,35.422,156.594
C09045=1070.912,428.420,-114.990,176.290,35.434,156.597
C09046=1070.921,428.666,-115.036,176.297,35.445,156.599
C09047=1070.929,428.912,-115.082,176.304,35.458,156.602
C09048=1070.937,429.157,-115.128,176.311,35.469,156.605
C09049=1070.945,429.403,-115.175,176.318,35.481,156.608
C09050=1070.954,429.648,-115.220,176.325,35.493,156.611
C09051=1070.962,429.894,-115.266,176.333,35.505,156.614
C09052=1070.971,430.140,-115.313,176.340,35.517,156.617
C09053=1070.978,430.385,-115.358,176.347,35.529,156.620
C09054=1070.987,430.630,-115.405,176.355,35.541,156.623
C09055=1070.996,430.876,-115.451,176.362,35.553,156.626
C09056=1071.004,431.122,-115.497,176.369,35.565,156.629
C09057=1071.012,431.367,-115.543,176.377,35.577,156.632
C09058=1071.020,431.613,-115.589,176.384,35.589,156.635
C09059=1071.029,431.858,-115.636,176.392,35.602,156.638
C09060=1071.038,432.104,-115.683,176.399,35.614,156.641
C09061=1071.045,432.349,-115.729,176.406,35.626,156.644
C09062=1071.054,432.594,-115.776,176.414,35.638,156.647
C09063=1071.063,432.840,-115.823,176.421,35.651,156.651
C09064=1071.071,433.085,-115.869,176.429,35.664,156.654
C09065=1071.080,433.331,-115.916,176.436,35.676,156.657
C09066=1071.088,433.576,-115.963,176.444,35.689,156.660
C09067=1071.096,433.821,-116.009,176.451,35.701,156.663
C09068=1071.105,434.066,-116.056,176.459,35.714,156.666
C09069=1071.113,434.312,-116.103,176.466,35.726,156.670
C09070=1071.121,434.558,-116.150,176.474,35.739,156.673
C09071=1071.130,434.803,-116.198,176.481,35.752,156.676
C09072=1071.138,435.048,-116.244,176.490,35.765,156.679
C09073=1071.147,435.294,-116.291,176.498,35.778,156.682
C09074=1071.156,435.539,-116.338,176.505,35.790,156.686
C09075=1071.164,435.784,-116.385,176.513,35.803,156.689
C09076=1071.173,436.030,-116.432,176.520,35.816,156.692
C09077=1071.182,436.275,-116.479,176.529,35.829,156.696
